(* CODESYS project ecomatDisplaytestIn2001.project
   Author: ifm electronic
   Version: 4.0.0.0
   Description: Project template for 4.3" ifm ecomat display  device with keypad.
   Title: ifm ecomatDisplay 4.3" 64bit with Keypad
   CompiledLibraryCompatibilityVersion: CODESYS V3.5 SP16 Patch 5
   Company: ifm electronic

Project tree, tasks and I/O mapping:
  Device : ecomatDisplay43inch_64bit, ifm electronic, version 3.5.19.72
    application Application
      libraries: ifm_ecomatDisplay43inch_Cnt, 1.1.0.0 (ifm electronic); ifmCANopenManager, * (ifm electronic); ifmRawCAN, * (ifm electronic); ifmBehavior, * (ifm electronic); ifmBehavior_ecomatDisplay, * (ifm electronic); ifmDevice_ecomatDisplay43inch, * (ifm electronic); ifmEcoSysLx_SysItf_Common, * (ifm electronic); ifmEcoSysLx_SysItf_Display, * (ifm electronic); ifmEcoSysLx_SysItf_IO, * (ifm electronic); ifmEcoSysLx_SysItf_Keypad, * (ifm electronic); ifmEcoSysLx_SysItf_Net, * (ifm electronic); ifmEcoSysLx_SysItf_Print, * (ifm electronic); ifmEcoSysLx_SysItf_RTC, * (ifm electronic); ifmEcoSysLx_SysItf_Service, * (ifm electronic); ifmEcoSysLx_SysItf_Storage, * (ifm electronic); ifmEcoSysLx_SysItf_SysInfo, * (ifm electronic); ifmEcoSysLx_SysItf_Touchscreen, * (ifm electronic); ifmFileUtil_ecomatDisplay, * (ifm electronic); ifmLLCAN, * (ifm electronic); ifmTypes, * (ifm electronic); ifmTypes_ecomatDisplay, * (ifm electronic); SM3_Basic, * (CODESYS); VisuSymbols, 4.5.0.0 (System); SysTimeCore, * (System); SysTimeRtc, * (System); SML_Basic, * (CODESYS); SM3_Ramps, * (3S - Smart Software Solutions GmbH); SysTypes Interfaces, * (System); Standard, 3.3.0.10 (System); Util, 3.5.19.0 (System); Standard64, 3.5.20.0 (System); BASIC, 3.31 (OSCAT); String Functions, 3.5.18.0 (3S - Smart Software Solutions GmbH)
      task VISU_TASK (cyclic, interval t#20ms, priority 15) calls VisuElems.Visu_Prg
      task Task (cyclic, interval 20 ms, priority 1) calls PLC_PRG
      task frame_control_1K500 (cyclic, interval t#20ms, priority 5) calls Main_FRAME_CONTROL
      GlobalVariables/
        global variables GVL_Buttons
        global variables GVL_PRG
        global variables GVL_KeyList
        global variables GVL_Sites
        Structs/
        global variables GVL_CAN
        global variables GVL_KeysConfig
        global variables Color
        data type ByteArray_t
      TextLists/
        text list TL_eKeyMapCodes
      image pool ifmImagePool
      FBs/
        location/
          function block locatoinSimulation [FBD]
        Paramater/
          function block TO_ArrayOfUsint [FBD]
          function block FB_ByteToBoolArray [FBD]
          function block FB_UpdatingDistanceParameter [FBD]
          function block parameterUpdate [FBD]
          function block PrepareParameterForCAN [FBD]
        Roboter_States/
          function block FB_CAN_TX_GetStates_Cyclic [FBD]
          function block FB_SoC_FromVoltage [ST]
        function block FB_DefineMotorControllerState [FBD]
        Controll/
          function block HMIControl [FBD]
          function block RoboterControl [FBD]
          function block AutomaticModeControl [FBD]
          function block SprayerControl [FBD]
        function block changeLanguage [FBD]
      image pool ImagePool
      Visu/
        visualisation Main_Site
        visualisation NewSiteFrame
        visualisation Srart_Site
        visualisation Roboter_Parameter
        visualisation Auto_Mode_Site
        visualisation Visu_Default
        visualisation keys_frame
        visualisation empty
      Programms/
        program PLC_PRG [FBD]: ACT_Errors_Handling, ACT_Setting, ACT_PressedKeysConfig, ACT_Button_Control
        program Main_FRAME_CONTROL [FBD]: ACT_FrameControl, ACT_RefreshhMI
      functions/
        function block FB_smoothCLK [FBD]
        function intToSelectOnBool [FBD]
        function block FB_CLK [FBD]
        function block Advanced_CTUD [FBD]
        function block fb_delay [FBD]
        function Stuffing_To_ArrayOfUsint [FBD]
        function F_AnyToByte [ST]
      can/
        function block FB_CAN_RX [FBD]
    Communication : Communication, ifm electronic, version 3.5.19.72
      Ethernet : Ethernet, ifm electronic, version 3.5.19.72
      CAN : CAN, ifm electronic, version 3.5.19.72
        CANbus : CANbus, ifm electronic, version 2.0.0.0
            settings: Baudrate = 500
  5ce3da45-db07-42e7-a21c-a00fff4ed8f6|E:\BSR\Me\May Be Useful\ifm-engg_Logo\IFMLO_PANT_2c.png
  5ce3da45-db07-42e7-a21c-a00fff4ed8f6|E:\BSR\OnSVN\CODESYS_V3x\PDM360-3\DesignDocs\Pictures\PDM Visu Templates 20181217\Bg_5Inch_dark.png
  5ce3da45-db07-42e7-a21c-a00fff4ed8f6|E:\BSR\OnSVN\CODESYS_V3x\PDM360-3\DesignDocs\Pictures\PDM Visu Templates 20181217\Bg_5Inch_lightPDM_Theming.png
  5ce3da45-db07-42e7-a21c-a00fff4ed8f6|E:\BSR\OnSVN\CODESYS_V3x\PDM360-3\DesignDocs\Pictures\PDM Visu Templates 20181217\Button_5Inch_dark.png
  5ce3da45-db07-42e7-a21c-a00fff4ed8f6|E:\BSR\OnSVN\CODESYS_V3x\PDM360-3\DesignDocs\Pictures\PDM Visu Templates 20181217\Button_5Inch_lightPDM_Theming.png
  5ce3da45-db07-42e7-a21c-a00fff4ed8f6|E:\BSR\OnSVN\CODESYS_V3x\PDM360-3\DesignDocs\Pictures\PDM Visu Templates 20181217\Button_And_Bg_5Inch_dark.png
  5ce3da45-db07-42e7-a21c-a00fff4ed8f6|E:\BSR\OnSVN\CODESYS_V3x\PDM360-3\DesignDocs\Pictures\PDM Visu Templates 20181217\Button_And_Bg_5Inch_lightPDM_Theming.png
  5ce3da45-db07-42e7-a21c-a00fff4ed8f6|C:\Users\indongpa\Downloads\Visu_KeyTemplates_ecomatDisplay43Inch_V2\LightBg_LightKey.png
  5ce3da45-db07-42e7-a21c-a00fff4ed8f6|C:\Users\indongpa\Downloads\Visu_KeyTemplates_ecomatDisplay43Inch_V2\WhiteBg_LightKey.png
  5ce3da45-db07-42e7-a21c-a00fff4ed8f6|C:\Users\indongpa\Downloads\Visu_Global_BG_ecomatDisplay43Inch_V1\Visu_Global_BG_NoKeys_ecomatDisplay43Inch.png
  5ce3da45-db07-42e7-a21c-a00fff4ed8f6|C:\Users\indongpa\OneDrive - ifm electronic gmbh\Downlaods\Visu_Global_BG_ecomatDisplay43Inch_V1\Visu_Global_BG_NoKeys_ecomatDisplay43Inch 90Deg.png
  5ce3da45-db07-42e7-a21c-a00fff4ed8f6|C:\Users\indongpa\Downloads\MicrosoftTeams-image (5).png
  5ce3da45-db07-42e7-a21c-a00fff4ed8f6|C:\Users\indongpa\Downloads\Visu_KeyTemplates_ecomatDisplay43Inch_V2\WhiteBg_DarkKey.png
  5ce3da45-db07-42e7-a21c-a00fff4ed8f6|C:\Users\indongpa\Downloads\Visu_Global_BG_ecomatDisplay43Inch_V1\Visu_Global_BG_WithKeys_ecomatDisplay43Inch.png
  5ce3da45-db07-42e7-a21c-a00fff4ed8f6|C:\Users\indongpa\Downloads\Visu_KeyTemplates_ecomatDisplay43Inch_V2\DarkBg_LightKey.png
  5ce3da45-db07-42e7-a21c-a00fff4ed8f6|C:\Users\indongpa\Downloads\Visu_KeyTemplates_ecomatDisplay43Inch_V2\Bg_Dark.png
  5ce3da45-db07-42e7-a21c-a00fff4ed8f6|C:\Users\indongpa\Downloads\Visu_KeyTemplates_ecomatDisplay43Inch_V2\Bg_Light.png
  Project Information/
    function GetCompany [ST]
    function GetTitle [ST]
    function GetVersion [ST]
    function GetTextProperty [ST]
    function GetTextProperty2 [ST]
    function GetNumberProperty [ST]
    function GetBooleanProperty [ST]
    function GetVersionProperty [ST]
  5ce3da45-db07-42e7-a21c-a00fff4ed8f6|C:\Users\indongpa\OneDrive - ifm electronic gmbh\Downlaods\Visu_Global_BG_ecomatDisplay43Inch_V1\Visu_Global_BG_WithKeys_ecomatDisplay43Inch 90Deg.png
  text list GlobalTextList
  5ce3da45-db07-42e7-a21c-a00fff4ed8f6|E:\BSR\Me\May Be Useful\ifm-engg_Logo\IFMLO_PANT_2c.png
  5ce3da45-db07-42e7-a21c-a00fff4ed8f6|C:\Users\indongpa\Downloads\Visu_KeyTemplates_ecomatDisplay43Inch_V2\DarkBg_LightKey.png
  5ce3da45-db07-42e7-a21c-a00fff4ed8f6|C:\Users\indongpa\Downloads\Visu_KeyTemplates_ecomatDisplay43Inch_V2\WhiteBg_DarkKey.png
  5ce3da45-db07-42e7-a21c-a00fff4ed8f6|C:\Users\indongpa\Downloads\Visu_KeyTemplates_ecomatDisplay43Inch_V2\LightBg_LightKey.png
  5ce3da45-db07-42e7-a21c-a00fff4ed8f6|C:\Users\indongpa\Downloads\Visu_KeyTemplates_ecomatDisplay43Inch_V2\WhiteBg_LightKey.png
  5ce3da45-db07-42e7-a21c-a00fff4ed8f6|C:\Users\indongpa\Downloads\Visu_Global_BG_ecomatDisplay43Inch_V1\Visu_Global_BG_WithKeys_ecomatDisplay43Inch.png
  5ce3da45-db07-42e7-a21c-a00fff4ed8f6|C:\Users\indongpa\OneDrive - ifm electronic gmbh\Downlaods\Visu_Global_BG_ecomatDisplay43Inch_V1\Visu_Global_BG_WithKeys_ecomatDisplay43Inch 90Deg.png
  5ce3da45-db07-42e7-a21c-a00fff4ed8f6|C:\Users\indongpa\Downloads\Visu_Global_BG_ecomatDisplay43Inch_V1\Visu_Global_BG_NoKeys_ecomatDisplay43Inch.png
  5ce3da45-db07-42e7-a21c-a00fff4ed8f6|C:\Users\indongpa\OneDrive - ifm electronic gmbh\Downlaods\Visu_Global_BG_ecomatDisplay43Inch_V1\Visu_Global_BG_NoKeys_ecomatDisplay43Inch 90Deg.png
  5ce3da45-db07-42e7-a21c-a00fff4ed8f6|C:\Users\indongpa\Downloads\Visu_KeyTemplates_ecomatDisplay43Inch_V2\Bg_Dark.png
  5ce3da45-db07-42e7-a21c-a00fff4ed8f6|C:\Users\indongpa\Downloads\Visu_KeyTemplates_ecomatDisplay43Inch_V2\Bg_Light.png
  5ce3da45-db07-42e7-a21c-a00fff4ed8f6|C:\Users\Administrator\Downloads\ant.png
  5ce3da45-db07-42e7-a21c-a00fff4ed8f6|C:\Users\Administrator\Downloads\Screenshot 2024-06-27 111636.png
  5ce3da45-db07-42e7-a21c-a00fff4ed8f6|C:\Users\Administrator\Downloads\Screenshot 2024-06-27 113436.png
  5ce3da45-db07-42e7-a21c-a00fff4ed8f6|C:\Users\moham\Downloads\splash_ant.bmp
  5ce3da45-db07-42e7-a21c-a00fff4ed8f6|C:\Users\Administrator\Downloads\ant_s.png
  5ce3da45-db07-42e7-a21c-a00fff4ed8f6|C:\Users\Administrator\Downloads\WhatsApp Image 2024-09-06 at 21.10.24.jpeg
  5ce3da45-db07-42e7-a21c-a00fff4ed8f6|C:\Users\Administrator\Downloads\battery fast Leer.png
  5ce3da45-db07-42e7-a21c-a00fff4ed8f6|C:\Users\Administrator\Downloads\images.jpg
  5ce3da45-db07-42e7-a21c-a00fff4ed8f6|C:\Users\Administrator\Downloads\304be42a-81d5-456b-8698-6dc5f69a8eec.jpg
  5ce3da45-db07-42e7-a21c-a00fff4ed8f6|C:\Users\Administrator\Downloads\269b2263-283b-4274-9266-790e9879ed38.jpg
  text list SwitchKeys
  5ce3da45-db07-42e7-a21c-a00fff4ed8f6|C:\Users\Administrator\Downloads\icons8-einstellung-50.png
  5ce3da45-db07-42e7-a21c-a00fff4ed8f6|C:\Users\Administrator\Downloads\battery_0.png
  5ce3da45-db07-42e7-a21c-a00fff4ed8f6|C:\Users\Administrator\Downloads\battery_10.png
  5ce3da45-db07-42e7-a21c-a00fff4ed8f6|C:\Users\Administrator\Downloads\battery_20.png
  5ce3da45-db07-42e7-a21c-a00fff4ed8f6|C:\Users\Administrator\Downloads\battery_30.png
  5ce3da45-db07-42e7-a21c-a00fff4ed8f6|C:\Users\Administrator\Downloads\battery_50.png
  5ce3da45-db07-42e7-a21c-a00fff4ed8f6|C:\Users\Administrator\Downloads\battery_70.png
  5ce3da45-db07-42e7-a21c-a00fff4ed8f6|C:\Users\Administrator\Downloads\battery_80.png
  5ce3da45-db07-42e7-a21c-a00fff4ed8f6|C:\Users\Administrator\Downloads\battery_90.png
  5ce3da45-db07-42e7-a21c-a00fff4ed8f6|C:\Users\Administrator\Downloads\battery_voll.png
  5ce3da45-db07-42e7-a21c-a00fff4ed8f6|C:\Users\moham\Downloads\ant(2).bmp
*)

// Device/Application/GlobalVariables/ByteArray_t
TYPE ByteArray_t : ARRAY[0..7] OF BYTE; END_TYPE

// Device/Application/GlobalVariables/GVL_Buttons
{attribute 'qualified_only'}
VAR_GLOBAL
	startAutoModeIsClicked: BOOL;
	stopAutoModeIsClicked: BOOL;
	//switschingToStartSite: BOOL;
	PauseAutoModeIsClicked: BOOL;
	backToStartScreenIsClicked: BOOL;
	settingClicked: BOOL;
	ResumeAutoModeIsClicked: BOOL;
	PauseOrResumeIsClicked: BOOL;
	
	
	// settings
		//time
		
// parameter
	//start time
	//sprayer
	sprayerUp : BOOL;
	sprayerDown : BOOL;
	sprayerLeft : BOOL;
	sprayerRight : BOOL;
	pump : BOOL;
	//Language
	englisch: BOOL;
	deutsch: BOOL;
	//changeHourClicked: BOOL;
	//changeMinuteClicked: BOOL;
END_VAR

// Device/Application/GlobalVariables/GVL_PRG
{attribute 'qualified_only'}
VAR_GLOBAL

	// HMI Mode
	deactivatePLCSimModeMan: BOOL;
	// visu frames control
	currentVisuFrame: INT := 0;
	refreshHMI : BOOL := FALSE; // use rising/falling trigger
	
	//parameter
	selectedParameterIndex: Int:= 0;
	bRowsDirection: BOOL;
	rCountRows: REAL;
	roboterWidth: REAL:= 0.5;
	dinstanceBetweenRowsMin: REAL := roboterWidth + 0.2; // m : min. distance between 2 Rows in meter. Ther is no max Value but the max Value is in CAN Frame for all distances d1,d2 and d3 = 12.8 m  
	turningDistancerMin: REAL:= 1.5; // min distance to be able to make a turn
	
	// Automode Control
	SR_autoMode: SR;
	RS_AM_Paused: RS;
	AM_Paused: BOOL;
	autoModestarted: BOOL;
	screenSwitching: BOOL;	// while switching the frame: true to disable all buttons
	enableAM : BOOL := TRUE;
	//State
	batteryState: USINT;
	enableStatesRequest : BOOL := TRUE;
	
	
	activate_FrameControl : BOOL := TRUE;
	
	//Sprayer
	
	enableSprayer : BOOL := TRUE;
	
	// CAN
	
	enableCanChannel_0: BOOL;
	canInfo: ifmTypes.DIAG_INFO;
	restartCan: BOOL;
	sprayerCanInfo: ifmTypes.DIAG_INFO;
	sprayerCanError: BOOL;
	canChannelError: BOOL;
	AM_CanFramError: BOOL;
	canError: BOOL;
	stetesCanError: BOOL;
	deactivateErrorHandling: BOOL;
	SR_startIsKlicked: SR;
	startMin: INT;
	startHour: INT;
	waitingStartTime: BOOL;
	simModeActive: BOOL;
	stopAM_Frame_received: BOOL;
	showkeys: BOOL;
	frameid: USINT;
	frameRefreshRequestCanError: BOOL;
	canFatalError: BOOL;
	fatalErrot: BOOL;
	to_am_frame: BOOL;
	stTime: ifmDevice.stDATE_TIME;
	acceleration: UINT;
	accelerationX10: UDINT;
	deceleration: UINT;
	decelerationX10: UDINT;
	settingCanError: BOOL;
	accelerationScreen: UINT;
	decelerationScreen: UINT;
END_VAR
VAR_GLOBAL RETAIN
	// setting
	language : STRING := 'EN';
	maxVoltage : REAL := 58.4;
	sprayerHight : REAL;
	MotorSpeed : USINT;
END_VAR
VAR_GLOBAL CONSTANT
		allwaysTrue : BOOL := TRUE;
END_VAR

// Device/Application/GlobalVariables/GVL_KeyList
{attribute 'qualified_only'}

(* 

!!! This GVL list is from project template !!!

The following variables are controlled by key events mapped at Default Hotkey mapping list in Visualization Manager.

For example, F1 function key of standard keyboard (MFII) is pressed, xF1 bit in this list will become TRUE; when the same 
key is released then xF1 become FALSE.

*)

VAR_GLOBAL

(* Display system key press / release event status. TRUE = Key Pressed, FALSE = Key Released  *)
	xF1 		: BOOL;		(* Event status of F1 function key *)
	xF2 		: BOOL;		(* Event status of F2 function key *)
	xF3 		: BOOL;		(* Event status of F3 function key *)
	xF4 		: BOOL;		(* Event status of F4 function key *)
	xF5 		: BOOL;		(* Event status of F5 function key *)
	xF6 		: BOOL;		(* Event status of F6 function key *)
	xF7 		: BOOL;		(* Event status of F7 function key *)
	xF8 		: BOOL;		(* Event status of F8 function key *)
	xF9 		: BOOL;		(* Event status of F9 function key *)
	xF10 		: BOOL;		(* Event status of F10 function key *)
	xUp 		: BOOL;		(* Event status of Up arrow key *)
	xDown		: BOOL;		(* Event status of Down arrow key *)
	xLeft 		: BOOL;		(* Event status of Left arrow key *)
	xRight 		: BOOL;		(* Event status of Right arrow key *)
	xKey_Return : BOOL;		(* Event status of Return (or Enter) key *)
END_VAR

// Device/Application/GlobalVariables/GVL_Sites
{attribute 'qualified_only'}
VAR_GLOBAL
	Parameter:STRING:= 'Roboter_Parameter';
	location: STRING:= 'LocationSeite_Inkrement';
END_VAR

// Device/Application/GlobalVariables/GVL_CAN
{attribute 'qualified_only'}
VAR_GLOBAL
	
	canChannnel: ifmDevice.CAN_CHANNEL := ifmDevice.CAN_CHANNEL.CHAN_0;
	// States ID 16x601
	getStatusState: ARRAY [0..7] OF USINT := [16#40,16#11,16#21,0,0,0,0,0];
	getFaultsState: ARRAY [0..7] OF USINT := [16#40,16#12,16#21,0,0,0,0,0];
	getBatteryState: ARRAY [0..7] OF USINT := [16#42,16#0D,16#21,2,0,0,0,0];
	getRuntimeStatus1: ARRAY [0..7] OF USINT := [16#40,16#22,16#21,1,0,0,0,0]; //1. Motor Andrew needs to change 1 and 2
	getRuntimeStatus2: ARRAY [0..7] OF USINT := [16#40,16#22,16#21,2,0,0,0,0]; //2. Motor
	
	// auto Mode
	automodeCanId: UDINT := 16#50;
	
	stop: ARRAY [0..7] OF USINT:=[255,0,0,0,0,0,0,0];
	pause: ARRAY [0..7] OF USINT:=[200,1,0,0,0,0,0,0];
	resume: ARRAY [0..7] OF USINT:=[200,2,0,0,0,0,0,0];
	
	// acceleration Profile
	//getAcceleration_1: ARRAY [0..7] OF USINT:=[16#40,16#83,16#60,1,0,0,0,0];
	//setAcceleration_1: ARRAY [0..7]OF USINT:=[16#40,16#83,16#60,1,0,0,0,0];
	//getDeceleration_1: ARRAY [0..7] OF USINT:=[16#40,16#84,16#60,1,0,0,0,0];
	//setDeceleration_1: ARRAY [0..7] OF USINT:=[16#40,16#07,16#20,1,0,0,0,0];
	
	//getAcceleration_2: ARRAY [0..7] OF USINT:=[16#40,16#83,16#60,1,0,0,0,0];
	//setAcceleration_2: ARRAY [0..7] OF USINT:=[16#40,16#08,16#20,1,0,0,0,0];
	//getDeceleration_2: ARRAY [0..7] OF USINT:=[16#40,16#84,16#60,1,0,0,0,0];
	//setDeceleration_2: ARRAY [0..7] OF USINT:=[16#40,16#07,16#20,1,0,0,0,0];
	//setAcceleration_1: ARRAY [0..7] OF USINT:=[16#40,16#08,16#20,1,0,0,0,0];
	
	// acceleration Value
	setAcceleration_1: ARRAY [0..7]OF USINT:=[16#23,16#06,16#20,1,0,0,0,0];
	setAcceleration_2: ARRAY [0..7]OF USINT:=[16#23,16#06,16#20,2,0,0,0,0];
	setDeceleration_1: ARRAY [0..7]OF USINT:=[16#23,16#07,16#20,1,0,0,0,0];
	setDeceleration_2: ARRAY [0..7]OF USINT:=[16#23,16#07,16#20,2,0,0,0,0];
	
	// max. rpm
	setRPM_max_1 :ARRAY [0..7]OF USINT:=[16#23,16#07,16#20,1,0,0,0,0];
	// get motors data
	reedRPM: ARRAY [0..7] OF USINT:=[16#40,16#03,16#21,1,0,0,0,0];// Min: -65535  Max: 65535
	Read_Battery_Amps : ARRAY [0..7] OF USINT:=[16#42,16#0C,16#21,1,0,0,0,0]; // Measures and reports the Amps flowing from the battery in Amps * 10
	Read_Battery_State_Of_Charge : ARRAY [0..7] OF USINT:=[16#42,16#3A,16#21,0,0,0,0,0]; // Battery state of charge in %
	//Sprayer
	
	motorcontrollerId: UDINT := 16#601;
	
	//control some of bits
	switchOffPump: ARRAY [0..7] OF USINT:=[16#2F,16#0A,16#20,0,6,0,0,0];
	switchOnPump: ARRAY [0..7] OF USINT:=[16#2F,16#09,16#20,0,6,0,0,0];
	switchOffSprayerLeft: ARRAY [0..7] OF USINT:=[16#2F,16#0A,16#20,0,7,0,0,0];
	switchOnSprayerLeft: ARRAY [0..7] OF USINT:=[16#2F,16#09,16#20,0,7,0,0,0];
	switchOffSprayerRight: ARRAY [0..7] OF USINT:=[16#2F,16#0A,16#20,0,8,0,0,0];
	switchOnSprayerRight: ARRAY [0..7] OF USINT:=[16#2F,16#09,16#20,0,8,0,0,0];
	sprayeStartUpFrame: ARRAY [0..7] OF USINT:=[47,9,32,0,2,0,0,0];// Andrew: 4->1 & -4->2 when paused & stop
	sprayerStopUpFrame: ARRAY [0..7] OF USINT:=[47,10,32,0,2,0,0,0];// When resume 4->1 & 2
	sprayerStartDownFrame: ARRAY [0..7] OF USINT:=[47,9,32,0,4,0,0,0];
	sprayerStopDownFrame: ARRAY [0..7] OF USINT:=[47,10,32,0,4,0,0,0];
	
	HMI_CAN_ID: UDINT := 16#19;
	ACK_Stop : ARRAY [0..7] OF USINT:=[3,0,0,0,0,0,0,0];
	stopFrameJetson : ARRAY [0..7] OF USINT :=[2,0,0,0,0,0,0,0];
	test: ARRAY [0..7] OF USINT := [8(1)];
END_VAR

// Device/Application/GlobalVariables/GVL_KeysConfig
{attribute 'qualified_only'}
VAR_GLOBAL
	countOfPressedKeys : USINT;
	oneKeyPressedForLongTime: BOOL;
	oneKeyOrMorePressed: BOOL;
	oneKeyPressed: BOOL;
	oneKeyPressedForLongTime_RT: BOOL;
END_VAR

// Device/Application/GlobalVariables/Color

{attribute 'qualified_only'}
VAR_GLOBAL
	
	NOT_DEFINED : DINT :=-1;
	Aqua : DINT :=16#FFFF;
	Black : DINT :=16#0;
	Blue : DINT :=16#FF;
	Brown : DINT :=16#A52A2A;
	Cyan : DINT :=16#FFFF;
	DarkBlue : DINT :=16#8B;
	DarkCyan : DINT :=16#8B8B;
	DarkGray : DINT :=16#A9A9A9;
	DarkGreen :DINT :=16#6400;
	DarkMagenta : DINT :=16#8B008B; 
	DarkRed : DINT :=16#8B0000;
	DimGray :DINT :=16#696969;
	Gray : DINT :=16#808080;
	Green : DINT :=16#8000;
	LightBlue : DINT :=16#ADD8E6;
	LightCyan : DINT :=16#E0FFFF;
	LightGray : DINT :=16#D3D3D3;
	LightGreen : DINT :=16#90EE90;
	LightYellow : DINT :=16#FFFFE0;
	Lime : DINT :=16#FF00;
	Magenta : DINT :=16#FF00FF;
	Maroon : DINT :=16#800000;
	Navy : DINT :=16#80;
	Olive : DINT :=16#808000;
	Purple : DINT :=16#800080;
	Red : DINT  :=16#FF0000;
	Silver : DINT :=16#C0C0C0;
	Teal : DINT :=16#8080;
	White : DINT :=16#FFFFFF;
	Yellow : DINT := 16#FFFF00;
	
	// Transperancy
	TRANSP_NO : BYTE := 16#FF;
	TRANSP_LOW : BYTE := 16#C0;
	TRANSP_MEDIUM : BYTE := 16#80;
	TRANSP_HIGH : BYTE := 16#40;
	TRANSP_FULL  : BYTE := 16#0;

	batteryColor : DINT := 16#8000;
	keysColor: UDINT := 16#FF6E00;

END_VAR

// Device/Application/Programms/PLC_PRG

(* !!! This POU is from project template !!! *)

PROGRAM PLC_PRG
VAR
	testframe: ARRAY [0..7] OF USINT := [16#40,16#11,16#21,0,0,0,0,0];
	canTestFrameTon : TON;
	RS_Test : RS;
	t_test : TIME := T#3000ms;
(* Below is the FB instance with initial values to set default key mapping. The default key map is as per the default values set for ifmDevice.stKEY_MAP_LIST. *)
	fbSetKeyMapping		: ifmDevice.SetKeyMapping;
	batteryStateInProcent: REAL;
	selectedParameterIndex: INT;
	FB_CAN_RX_0: FB_CAN_RX;
	FB_CAN_TX_GetStates_Cyclic_0: FB_CAN_TX_GetStates_Cyclic;
	FB_HMIControl_0: HMIControl;
	getUpdatedParameter: parameterUpdate;
	RoboterautoModeControl_0: RoboterControl;
	SprayerControl_0: SprayerControl;
	//locatoinSimulation_0: locatoinSimulation;
	CAN_Tx_0: ifmRCAN.CAN_Tx;

	keyDelay: TON := (PT := TIME#300MS);

	goToParameterFrame: BOOL;
	
	// ERRORS handling
	RS_DisableCan: Standard.RS;
	TON_CanDisabled: Standard.TON ;
	test: BOOL;
	ctu_restart_counter: Standard.CTU;
	SR_simModeActive: SR;
	usiNumberRetryCanRecover: USINT := 5;
	rs_canrec: rs;
	restartRecovery: BOOL;
	testAfterRecover: FB_clk;
	resetErrors: BOOL;
	Advanced_CTUD_changeSysTimeMin: Advanced_CTUD;
	Advanced_CTUD_changeSysTimeHour: Advanced_CTUD;
	test2: UINT;
	test3: ByteArray_t;
	acceleration: UDINT;
	ChangingAcceleration_0: Advanced_CTUD;
	CAN_Tx_setAcceleration_1: ifmRCAN.CAN_Tx;
	ChangingDeceleration_0: Advanced_CTUD;
	CAN_Tx_setDeceleration_1: ifmRCAN.CAN_Tx;
	CAN_Tx_setDeceleration_2: ifmRCAN.CAN_Tx;
	CAN_Tx_setAcceleration_2: ifmRCAN.CAN_Tx;
	TON_F1: TON;
	TON_F3: TON;
END_VAR
// setting
VAR
	currentSettingFrameId : SINT := 0;
	//currentMaxRows : USINT := 0;

	//countOfSeconderyMeneuRows2 : ARRAY [0 .. countOfSettingRows] OF SINT:= [0,0,1];
	//
	//EN: BOOL ;
	DE : BOOL ;
	RO : BOOL ;
	changeLanguage_EN: changeLanguage;
	changeLanguage_DE: changeLanguage;
	//mainMeneuActive : BOOL := TRUE;
	
	SR_DeactivateLeftMeneu: SR;
	deactivateMainMeneu: BOOL;
	deactivateSeconderyMeneu: BOOL;
	selectedRowNum_Right: SINT := 0;//-1;
	selectedRowNum_left: SINT  := 0;//-1;
	SR_Enable: SR;
	enable: BOOL := TRUE;
	SR_activate3rdColumn: SR;
	thirdColumnActive: BOOL;
	visuhelp : BOOL;
	TON_Delay: TON := (PT := TIME#105ms);
	selectedRowNum_Right2: SINT;
	RS_visuHelp2: RS;
	RS_visuHelp3: RS;
	RS_visuHelp4: RS;
	pumpOn: BOOL;
	RS_pump: RS;
	sprayerSelectionLimit: SINT;
	languageselectionLimit : SINT;
	TOGGLE_Pump: TOGGLE;
	hourSetting: UINT;
	settedHoursNow: UINT;
	setTime: BOOL;
	SetSysTime: ifmDevice.SetSysTime;
	newTime: ifmDevice.stDATE_TIME;
	CAN_Recover_0 : ifmRCAN.CAN_Recover;
END_VAR
VAR CONSTANT
	countOfSettingRows: SINT := 1;
	sprayerId : USINT := 1;
	languageID : USINT := 0;
	timeId: USINT := 2;
	countOfSeconderyMeneuRows : ARRAY [0 .. countOfSettingRows] OF SINT:= [1,4];
END_VAR

//button control
VAR
	startTime : TIME_OF_DAY;
	TON_StopresumeButtonVisible: ton;
	StopresumeButtonVisible: BOOL;
END_VAR
VAR // added by the converter: edge detectors and wires of the graphical bodies
    _rt1, _rt2, _rt3, _rt4, _rt5, _rt6, _rt7, _rt8, _rt9, _rt10, _rt11, _rt12, _rt13, _rt14, _rt15, _rt16, _rt17, _rt18, _rt19, _rt20, _rt21, _rt22, _rt23, _rt24, _rt25 : R_TRIG;
    _ft1, _ft2, _ft3, _ft4, _ft5, _ft6, _ft7, _ft8 : F_TRIG;
    _w1, _w2, _w3 : BOOL;
    _w4, _w5, _w6, _w7, _w8, _w9, _w10, _w11 : USINT;
END_VAR

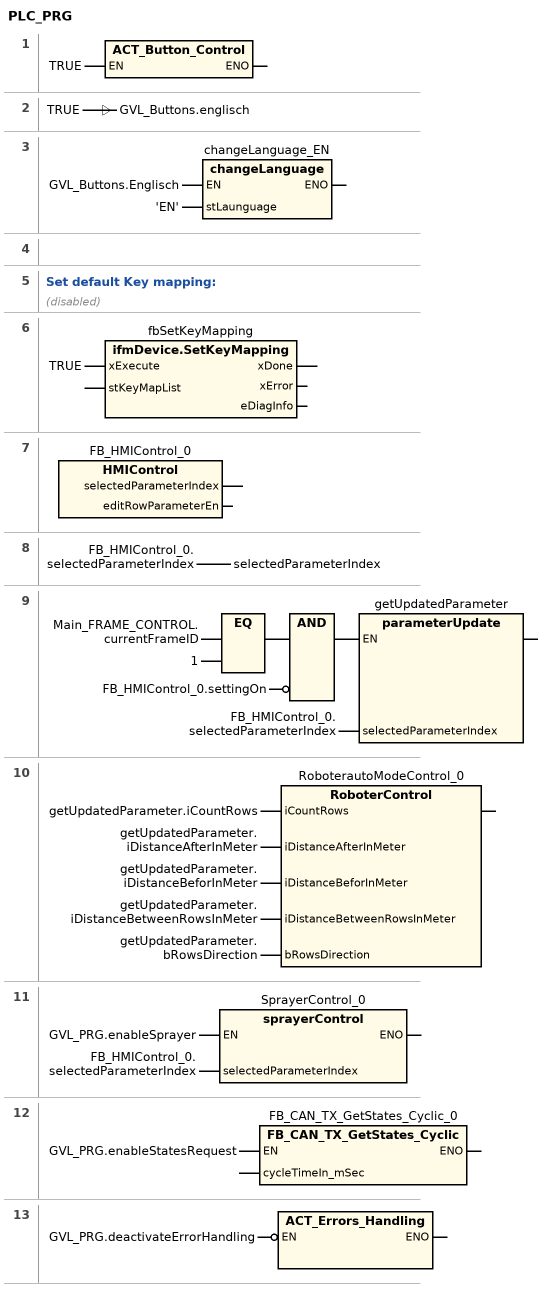
// NETWORK 1
ACT_Button_Control();

// NETWORK 2
_rt1(CLK := TRUE);
GVL_Buttons.englisch := _rt1.Q;

// NETWORK 3
IF GVL_Buttons.Englisch THEN
    changeLanguage_EN(stLaunguage := 'EN'); // changeLanguage
END_IF

// NETWORK 4

// NETWORK 5 (disabled)
// label: Set default Key mapping

// NETWORK 6
fbSetKeyMapping(xExecute := TRUE); // ifmDevice.SetKeyMapping

// NETWORK 7
FB_HMIControl_0(); // HMIControl

// NETWORK 8
selectedParameterIndex := FB_HMIControl_0.selectedParameterIndex;

// NETWORK 9
getUpdatedParameter(EN := Main_FRAME_CONTROL.currentFrameID = 1 AND NOT FB_HMIControl_0.settingOn, selectedParameterIndex := FB_HMIControl_0.selectedParameterIndex); // parameterUpdate

// NETWORK 10
RoboterautoModeControl_0(
    iCountRows := getUpdatedParameter.iCountRows,
    iDistanceAfterInMeter := getUpdatedParameter.iDistanceAfterInMeter,
    iDistanceBeforInMeter := getUpdatedParameter.iDistanceBeforInMeter,
    iDistanceBetweenRowsInMeter := getUpdatedParameter.iDistanceBetweenRowsInMeter,
    bRowsDirection := getUpdatedParameter.bRowsDirection); // RoboterControl

// NETWORK 11
IF GVL_PRG.enableSprayer THEN
    SprayerControl_0(selectedParameterIndex := FB_HMIControl_0.selectedParameterIndex); // sprayerControl
END_IF

// NETWORK 12
IF GVL_PRG.enableStatesRequest THEN
    FB_CAN_TX_GetStates_Cyclic_0(); // FB_CAN_TX_GetStates_Cyclic
END_IF

// NETWORK 13
IF NOT GVL_PRG.deactivateErrorHandling THEN ACT_Errors_Handling(); END_IF

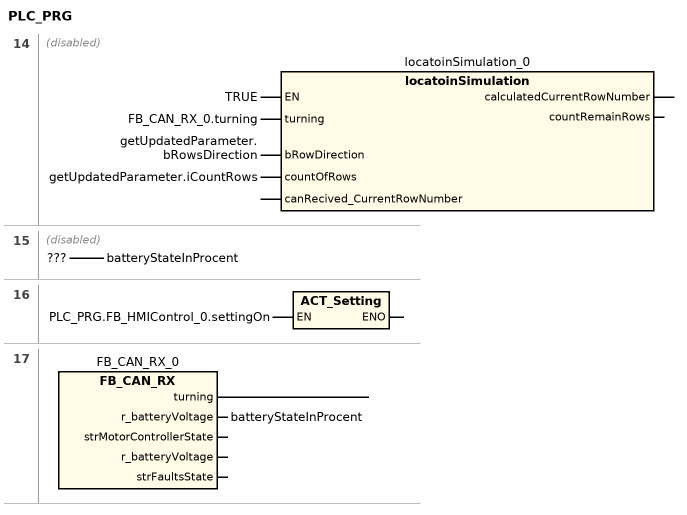
// NETWORK 14 (disabled)
// locatoinSimulation_0(
//     EN := TRUE,
//     turning := FB_CAN_RX_0.turning,
//     bRowDirection := getUpdatedParameter.bRowsDirection,
//     countOfRows := getUpdatedParameter.iCountRows); // locatoinSimulation

// NETWORK 15 (disabled)
// batteryStateInProcent := ???;

// NETWORK 16
IF PLC_PRG.FB_HMIControl_0.settingOn THEN ACT_Setting(); END_IF

// NETWORK 17
FB_CAN_RX_0(r_batteryVoltage => batteryStateInProcent); // FB_CAN_RX

ACTION ACT_Errors_Handling:
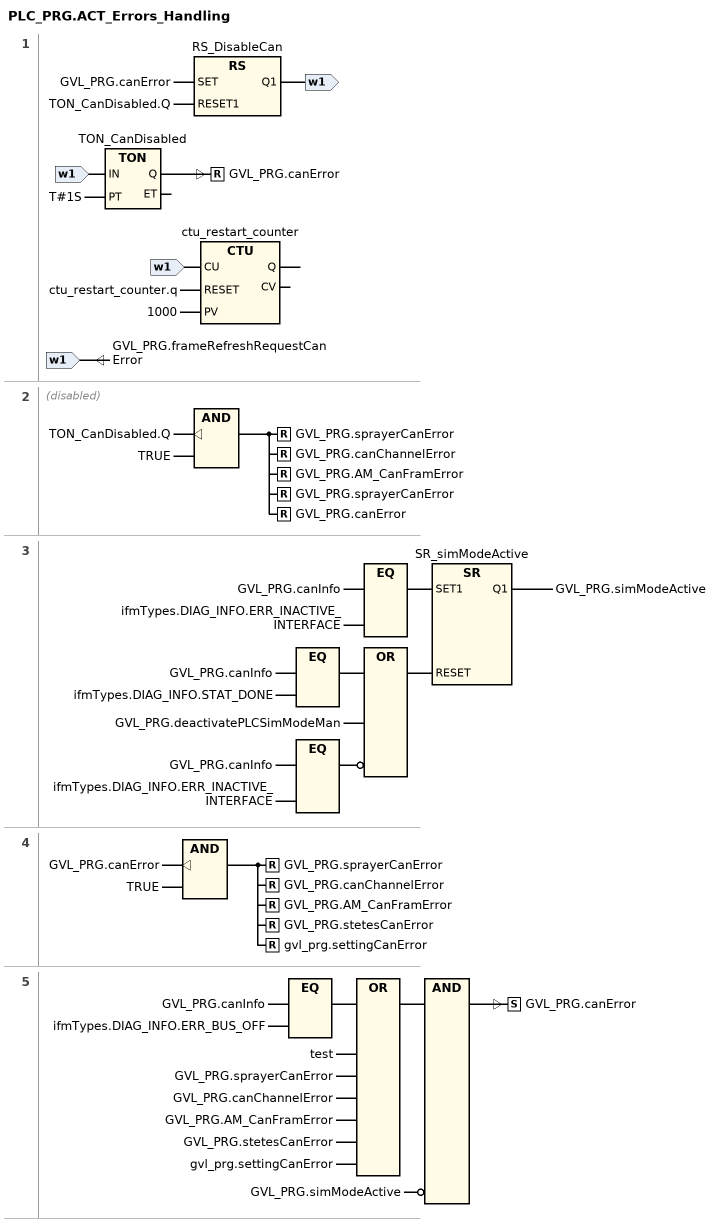
// NETWORK 1
RS_DisableCan(SET := GVL_PRG.canError, RESET1 := TON_CanDisabled.Q); // RS
TON_CanDisabled(IN := RS_DisableCan.Q1, PT := T#1S); // TON
_rt2(CLK := TON_CanDisabled.Q);
GVL_PRG.canError R= _rt2.Q;
ctu_restart_counter(CU := RS_DisableCan.Q1, RESET := ctu_restart_counter.q, PV := 1000); // CTU
_ft1(CLK := RS_DisableCan.Q1);
GVL_PRG.frameRefreshRequestCanError := _ft1.Q;

// NETWORK 2 (disabled)
// _ft2(CLK := TON_CanDisabled.Q);
// _w1 := _ft2.Q AND TRUE;
// GVL_PRG.sprayerCanError R= _w1;
// GVL_PRG.canChannelError R= _w1;
// GVL_PRG.AM_CanFramError R= _w1;
// GVL_PRG.sprayerCanError R= _w1;
// GVL_PRG.canError R= _w1;

// NETWORK 3
SR_simModeActive(SET1 := GVL_PRG.canInfo = ifmTypes.DIAG_INFO.ERR_INACTIVE_INTERFACE, RESET := GVL_PRG.canInfo = ifmTypes.DIAG_INFO.STAT_DONE OR GVL_PRG.deactivatePLCSimModeMan OR NOT (GVL_PRG.canInfo = ifmTypes.DIAG_INFO.ERR_INACTIVE_INTERFACE)); // SR
GVL_PRG.simModeActive := SR_simModeActive.Q1;

// NETWORK 4
_ft3(CLK := GVL_PRG.canError);
_w2 := _ft3.Q AND TRUE;
GVL_PRG.sprayerCanError R= _w2;
GVL_PRG.canChannelError R= _w2;
GVL_PRG.AM_CanFramError R= _w2;
GVL_PRG.stetesCanError R= _w2;
gvl_prg.settingCanError R= _w2;

// NETWORK 5
_rt3(CLK := (GVL_PRG.canInfo = ifmTypes.DIAG_INFO.ERR_BUS_OFF OR test OR GVL_PRG.sprayerCanError OR GVL_PRG.canChannelError OR GVL_PRG.AM_CanFramError OR GVL_PRG.stetesCanError OR gvl_prg.settingCanError) AND NOT GVL_PRG.simModeActive);
GVL_PRG.canError S= _rt3.Q;

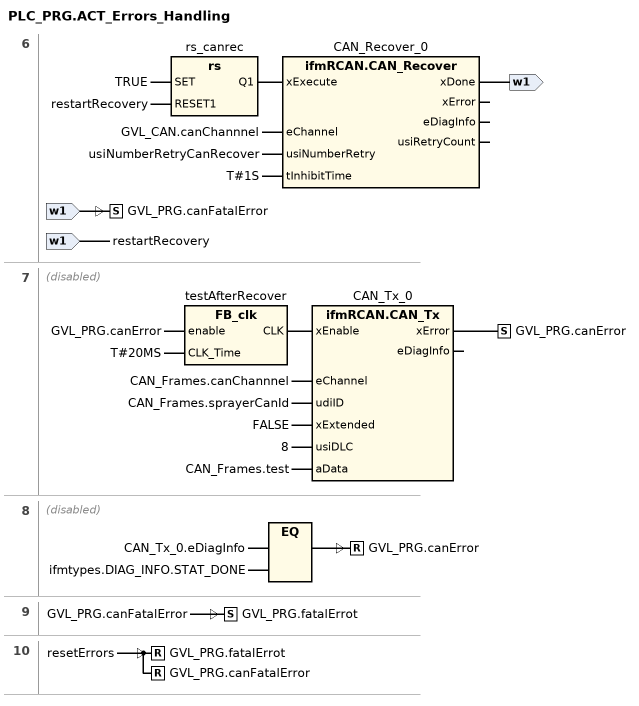
// NETWORK 6
rs_canrec(SET := TRUE, RESET1 := restartRecovery); // rs
CAN_Recover_0(
    xExecute := rs_canrec.Q1,
    eChannel := GVL_CAN.canChannnel,
    usiNumberRetry := usiNumberRetryCanRecover,
    tInhibitTime := T#1S); // ifmRCAN.CAN_Recover
_rt4(CLK := CAN_Recover_0.xDone);
GVL_PRG.canFatalError S= _rt4.Q;
restartRecovery := CAN_Recover_0.xDone;

// NETWORK 7 (disabled)
// testAfterRecover(enable := GVL_PRG.canError, CLK_Time := T#20MS); // FB_clk
// CAN_Tx_0(
//     xEnable := testAfterRecover.CLK,
//     eChannel := CAN_Frames.canChannnel,
//     udiID := CAN_Frames.sprayerCanId,
//     xExtended := FALSE,
//     usiDLC := 8,
//     aData := CAN_Frames.test); // ifmRCAN.CAN_Tx
// GVL_PRG.canError S= CAN_Tx_0.xError;

// NETWORK 8 (disabled)
// _rt5(CLK := CAN_Tx_0.eDiagInfo = ifmtypes.DIAG_INFO.STAT_DONE);
// GVL_PRG.canError R= _rt5.Q;

// NETWORK 9
_rt6(CLK := GVL_PRG.canFatalError);
GVL_PRG.fatalErrot S= _rt6.Q;

// NETWORK 10
_rt7(CLK := resetErrors);
GVL_PRG.fatalErrot R= _rt7.Q;
GVL_PRG.canFatalError R= _rt7.Q;
END_ACTION

ACTION ACT_Setting:
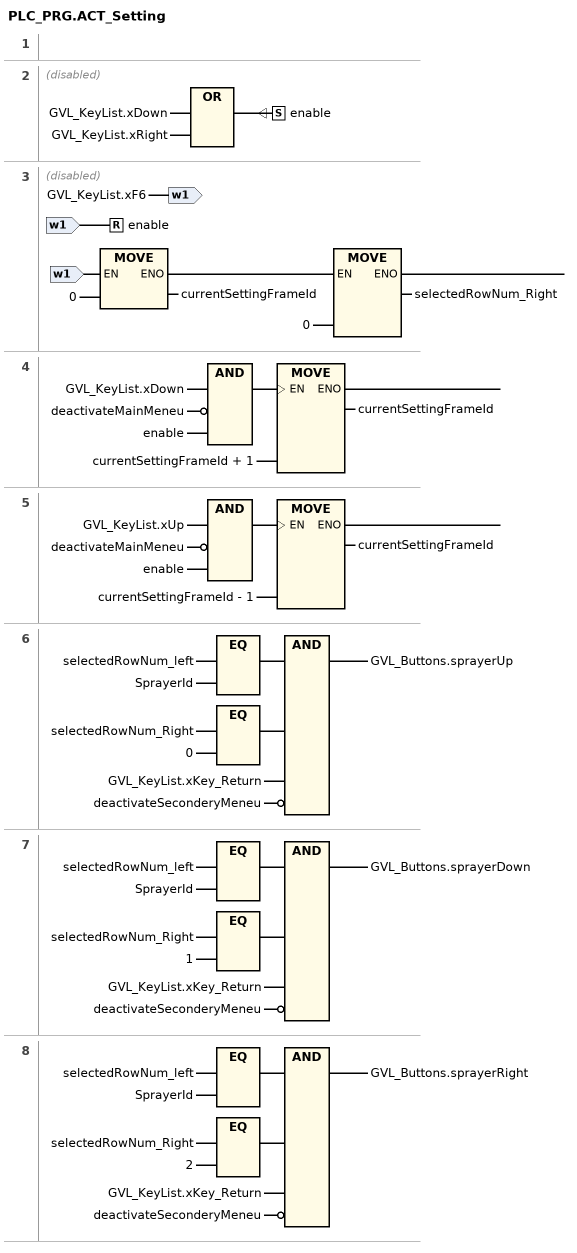
// NETWORK 1

// NETWORK 2 (disabled)
// _ft4(CLK := GVL_KeyList.xDown OR GVL_KeyList.xRight);
// enable S= _ft4.Q;

// NETWORK 3 (disabled)
// _rt8(CLK := GVL_KeyList.xF6);
// enable R= _rt8.Q;
// _w3 := _rt8.Q;
// IF _w3 THEN currentSettingFrameId := 0; END_IF
// IF _w3 THEN selectedRowNum_Right := 0; END_IF

// NETWORK 4
_rt9(CLK := GVL_KeyList.xDown AND NOT deactivateMainMeneu AND enable);
IF _rt9.Q THEN currentSettingFrameId := currentSettingFrameId + 1; END_IF

// NETWORK 5
_rt10(CLK := GVL_KeyList.xUp AND NOT deactivateMainMeneu AND enable);
IF _rt10.Q THEN currentSettingFrameId := currentSettingFrameId - 1; END_IF

// NETWORK 6
GVL_Buttons.sprayerUp := selectedRowNum_left = SprayerId AND selectedRowNum_Right = 0 AND GVL_KeyList.xKey_Return AND NOT deactivateSeconderyMeneu;

// NETWORK 7
GVL_Buttons.sprayerDown := selectedRowNum_left = SprayerId AND selectedRowNum_Right = 1 AND GVL_KeyList.xKey_Return AND NOT deactivateSeconderyMeneu;

// NETWORK 8
GVL_Buttons.sprayerRight := selectedRowNum_left = SprayerId AND selectedRowNum_Right = 2 AND GVL_KeyList.xKey_Return AND NOT deactivateSeconderyMeneu;

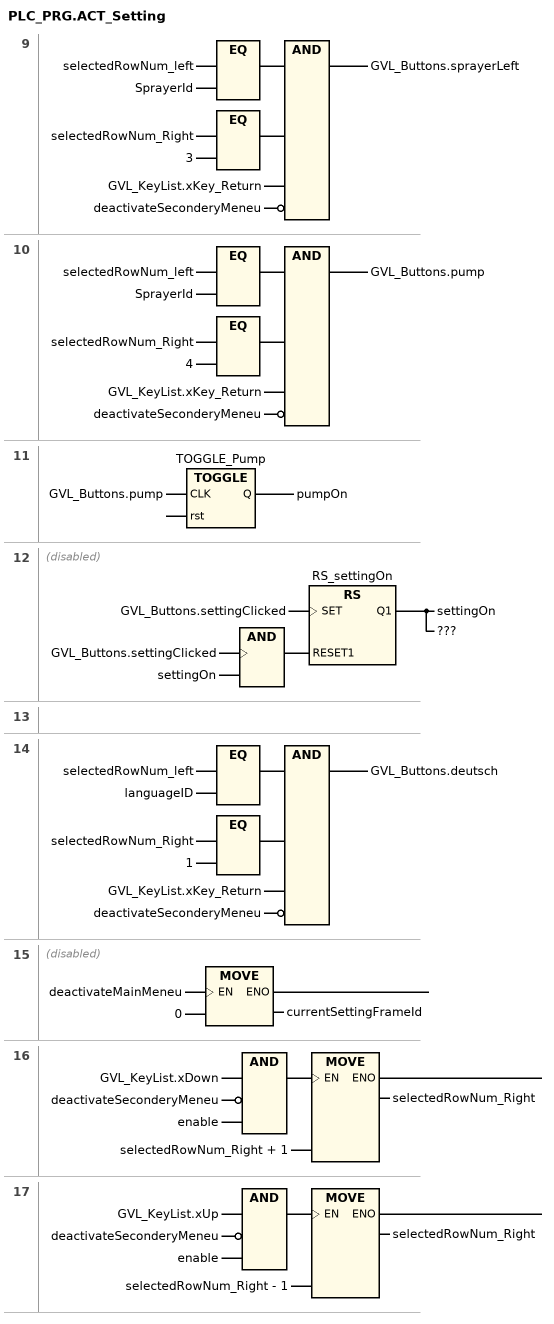
// NETWORK 9
GVL_Buttons.sprayerLeft := selectedRowNum_left = SprayerId AND selectedRowNum_Right = 3 AND GVL_KeyList.xKey_Return AND NOT deactivateSeconderyMeneu;

// NETWORK 10
GVL_Buttons.pump := selectedRowNum_left = SprayerId AND selectedRowNum_Right = 4 AND GVL_KeyList.xKey_Return AND NOT deactivateSeconderyMeneu;

// NETWORK 11
TOGGLE_Pump(CLK := GVL_Buttons.pump); // TOGGLE
pumpOn := TOGGLE_Pump.Q;

// NETWORK 12 (disabled)
// _rt11(CLK := GVL_Buttons.settingClicked);
// _rt12(CLK := GVL_Buttons.settingClicked);
// RS_settingOn(SET := _rt11.Q, RESET1 := _rt12.Q AND settingOn); // RS
// settingOn := RS_settingOn.Q1;
// ??? := RS_settingOn.Q1;

// NETWORK 13

// NETWORK 14
GVL_Buttons.deutsch := selectedRowNum_left = languageID AND selectedRowNum_Right = 1 AND GVL_KeyList.xKey_Return AND NOT deactivateSeconderyMeneu;

// NETWORK 15 (disabled)
// _rt13(CLK := deactivateMainMeneu);
// IF _rt13.Q THEN currentSettingFrameId := 0; END_IF

// NETWORK 16
_rt14(CLK := GVL_KeyList.xDown AND NOT deactivateSeconderyMeneu AND enable);
IF _rt14.Q THEN selectedRowNum_Right := selectedRowNum_Right + 1; END_IF

// NETWORK 17
_rt15(CLK := GVL_KeyList.xUp AND NOT deactivateSeconderyMeneu AND enable);
IF _rt15.Q THEN selectedRowNum_Right := selectedRowNum_Right - 1; END_IF

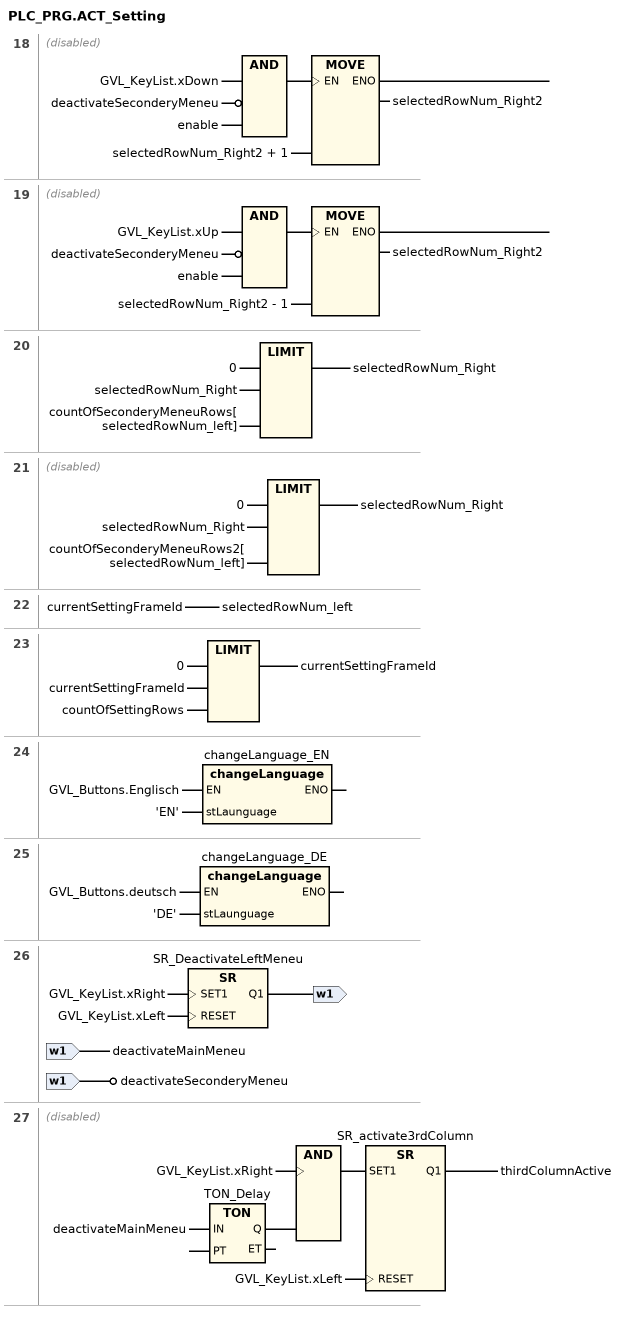
// NETWORK 18 (disabled)
// _rt16(CLK := GVL_KeyList.xDown AND NOT deactivateSeconderyMeneu AND enable);
// IF _rt16.Q THEN selectedRowNum_Right2 := selectedRowNum_Right2 + 1; END_IF

// NETWORK 19 (disabled)
// _rt17(CLK := GVL_KeyList.xUp AND NOT deactivateSeconderyMeneu AND enable);
// IF _rt17.Q THEN selectedRowNum_Right2 := selectedRowNum_Right2 - 1; END_IF

// NETWORK 20
selectedRowNum_Right := LIMIT(0, selectedRowNum_Right, countOfSeconderyMeneuRows[selectedRowNum_left]);

// NETWORK 21 (disabled)
// selectedRowNum_Right := LIMIT(0, selectedRowNum_Right, countOfSeconderyMeneuRows2[selectedRowNum_left]);

// NETWORK 22
selectedRowNum_left := currentSettingFrameId;

// NETWORK 23
currentSettingFrameId := LIMIT(0, currentSettingFrameId, countOfSettingRows);

// NETWORK 24
IF GVL_Buttons.Englisch THEN
    changeLanguage_EN(stLaunguage := 'EN'); // changeLanguage
END_IF

// NETWORK 25
IF GVL_Buttons.deutsch THEN
    changeLanguage_DE(stLaunguage := 'DE'); // changeLanguage
END_IF

// NETWORK 26
_rt18(CLK := GVL_KeyList.xRight);
_rt19(CLK := GVL_KeyList.xLeft);
SR_DeactivateLeftMeneu(SET1 := _rt18.Q, RESET := _rt19.Q); // SR
deactivateMainMeneu := SR_DeactivateLeftMeneu.Q1;
deactivateSeconderyMeneu := NOT SR_DeactivateLeftMeneu.Q1;

// NETWORK 27 (disabled)
// _rt20(CLK := GVL_KeyList.xRight);
// TON_Delay(IN := deactivateMainMeneu); // TON
// _rt21(CLK := GVL_KeyList.xLeft);
// SR_activate3rdColumn(SET1 := _rt20.Q AND TON_Delay.Q, RESET := _rt21.Q); // SR
// thirdColumnActive := SR_activate3rdColumn.Q1;

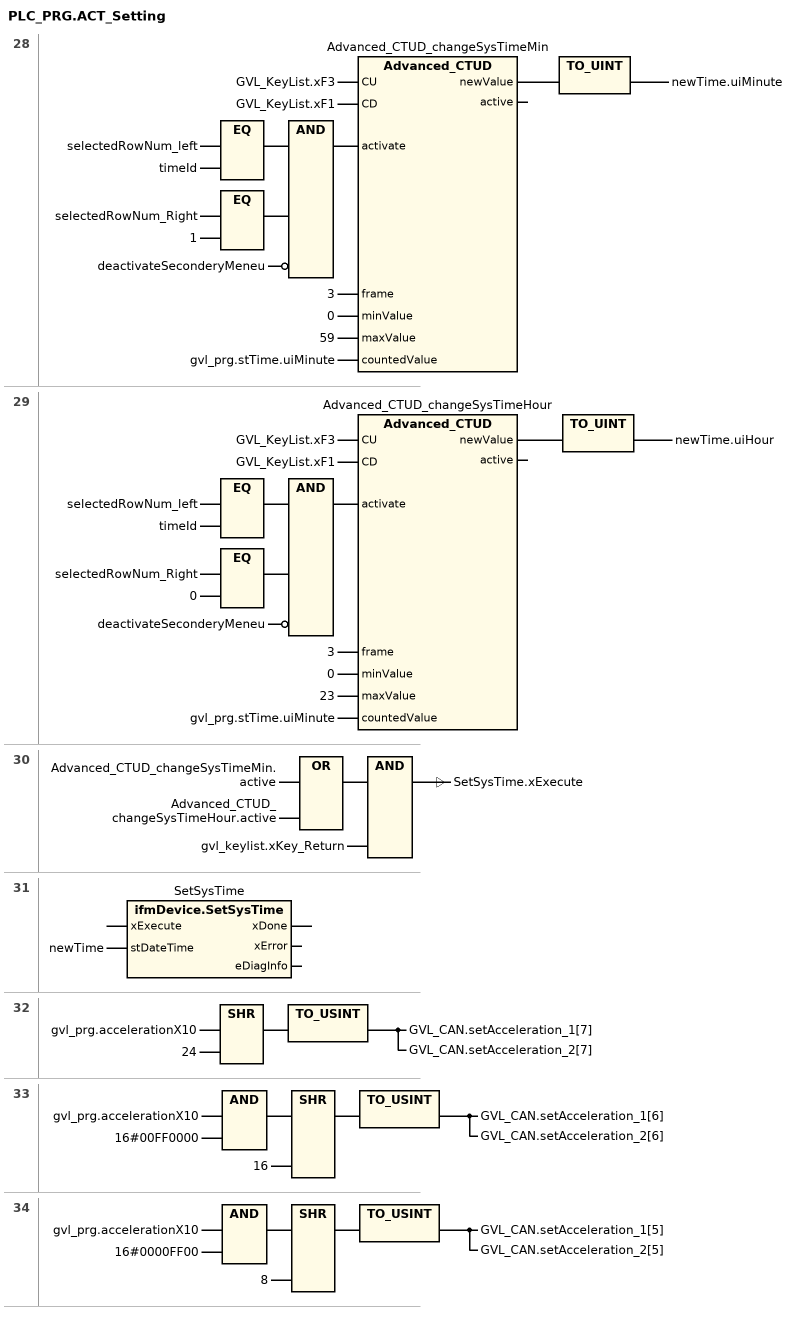
// NETWORK 28
Advanced_CTUD_changeSysTimeMin(
    CU := GVL_KeyList.xF3,
    CD := GVL_KeyList.xF1,
    activate := selectedRowNum_left = timeId AND selectedRowNum_Right = 1 AND NOT deactivateSeconderyMeneu,
    frame := 3,
    minValue := 0,
    maxValue := 59,
    countedValue := gvl_prg.stTime.uiMinute); // Advanced_CTUD
newTime.uiMinute := TO_UINT(Advanced_CTUD_changeSysTimeMin.newValue);

// NETWORK 29
Advanced_CTUD_changeSysTimeHour(
    CU := GVL_KeyList.xF3,
    CD := GVL_KeyList.xF1,
    activate := selectedRowNum_left = timeId AND selectedRowNum_Right = 0 AND NOT deactivateSeconderyMeneu,
    frame := 3,
    minValue := 0,
    maxValue := 23,
    countedValue := gvl_prg.stTime.uiMinute); // Advanced_CTUD
newTime.uiHour := TO_UINT(Advanced_CTUD_changeSysTimeHour.newValue);

// NETWORK 30
_rt22(CLK := (Advanced_CTUD_changeSysTimeMin.active OR Advanced_CTUD_changeSysTimeHour.active) AND gvl_keylist.xKey_Return);
SetSysTime.xExecute := _rt22.Q;

// NETWORK 31
SetSysTime(stDateTime := newTime); // ifmDevice.SetSysTime

// NETWORK 32
_w4 := TO_USINT(SHR(gvl_prg.accelerationX10, 24));
GVL_CAN.setAcceleration_1[7] := _w4;
GVL_CAN.setAcceleration_2[7] := _w4;

// NETWORK 33
_w5 := TO_USINT(SHR(gvl_prg.accelerationX10 AND 16#00FF0000, 16));
GVL_CAN.setAcceleration_1[6] := _w5;
GVL_CAN.setAcceleration_2[6] := _w5;

// NETWORK 34
_w6 := TO_USINT(SHR(gvl_prg.accelerationX10 AND 16#0000FF00, 8));
GVL_CAN.setAcceleration_1[5] := _w6;
GVL_CAN.setAcceleration_2[5] := _w6;

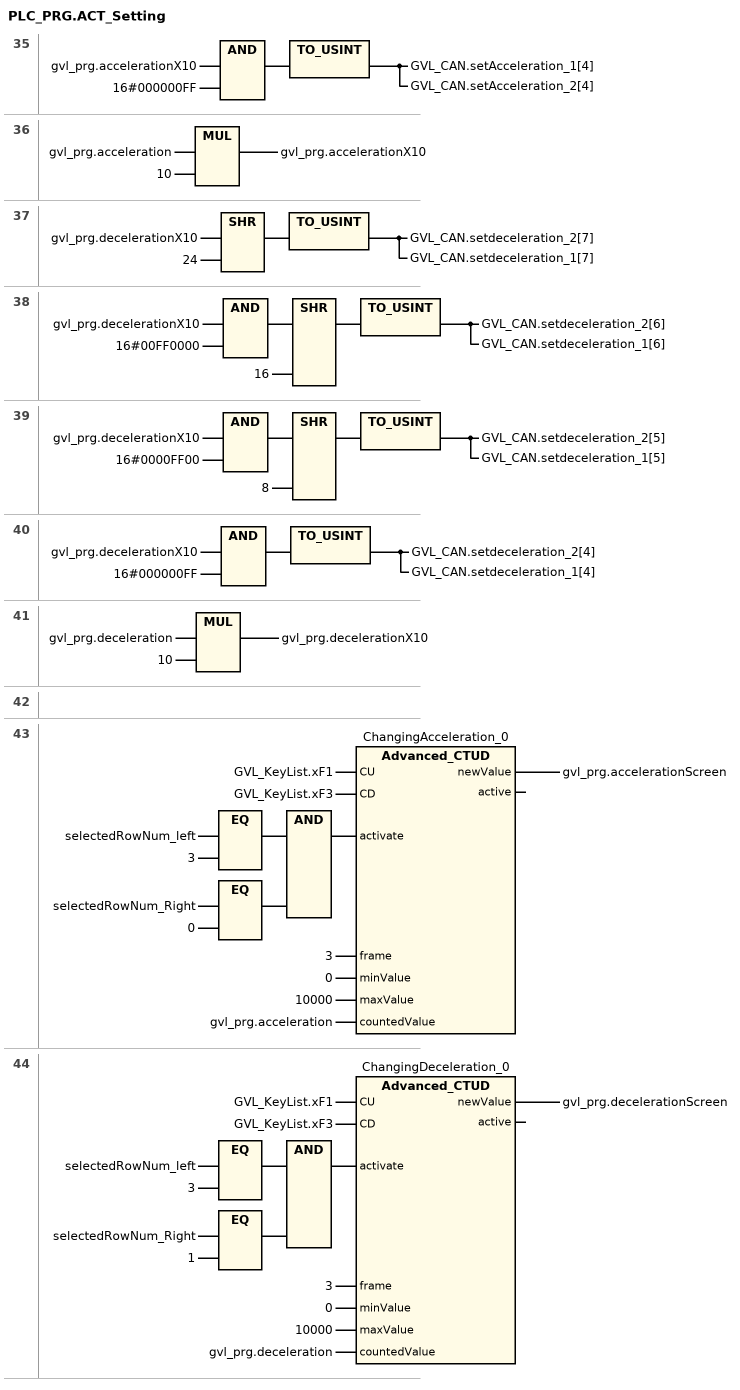
// NETWORK 35
_w7 := TO_USINT(gvl_prg.accelerationX10 AND 16#000000FF);
GVL_CAN.setAcceleration_1[4] := _w7;
GVL_CAN.setAcceleration_2[4] := _w7;

// NETWORK 36
gvl_prg.accelerationX10 := gvl_prg.acceleration * 10;

// NETWORK 37
_w8 := TO_USINT(SHR(gvl_prg.decelerationX10, 24));
GVL_CAN.setdeceleration_2[7] := _w8;
GVL_CAN.setdeceleration_1[7] := _w8;

// NETWORK 38
_w9 := TO_USINT(SHR(gvl_prg.decelerationX10 AND 16#00FF0000, 16));
GVL_CAN.setdeceleration_2[6] := _w9;
GVL_CAN.setdeceleration_1[6] := _w9;

// NETWORK 39
_w10 := TO_USINT(SHR(gvl_prg.decelerationX10 AND 16#0000FF00, 8));
GVL_CAN.setdeceleration_2[5] := _w10;
GVL_CAN.setdeceleration_1[5] := _w10;

// NETWORK 40
_w11 := TO_USINT(gvl_prg.decelerationX10 AND 16#000000FF);
GVL_CAN.setdeceleration_2[4] := _w11;
GVL_CAN.setdeceleration_1[4] := _w11;

// NETWORK 41
gvl_prg.decelerationX10 := gvl_prg.deceleration * 10;

// NETWORK 42

// NETWORK 43
ChangingAcceleration_0(
    CU := GVL_KeyList.xF1,
    CD := GVL_KeyList.xF3,
    activate := selectedRowNum_left = 3 AND selectedRowNum_Right = 0,
    frame := 3,
    minValue := 0,
    maxValue := 10000,
    countedValue := gvl_prg.acceleration); // Advanced_CTUD
gvl_prg.accelerationScreen := ChangingAcceleration_0.newValue;

// NETWORK 44
ChangingDeceleration_0(
    CU := GVL_KeyList.xF1,
    CD := GVL_KeyList.xF3,
    activate := selectedRowNum_left = 3 AND selectedRowNum_Right = 1,
    frame := 3,
    minValue := 0,
    maxValue := 10000,
    countedValue := gvl_prg.deceleration); // Advanced_CTUD
gvl_prg.decelerationScreen := ChangingDeceleration_0.newValue;

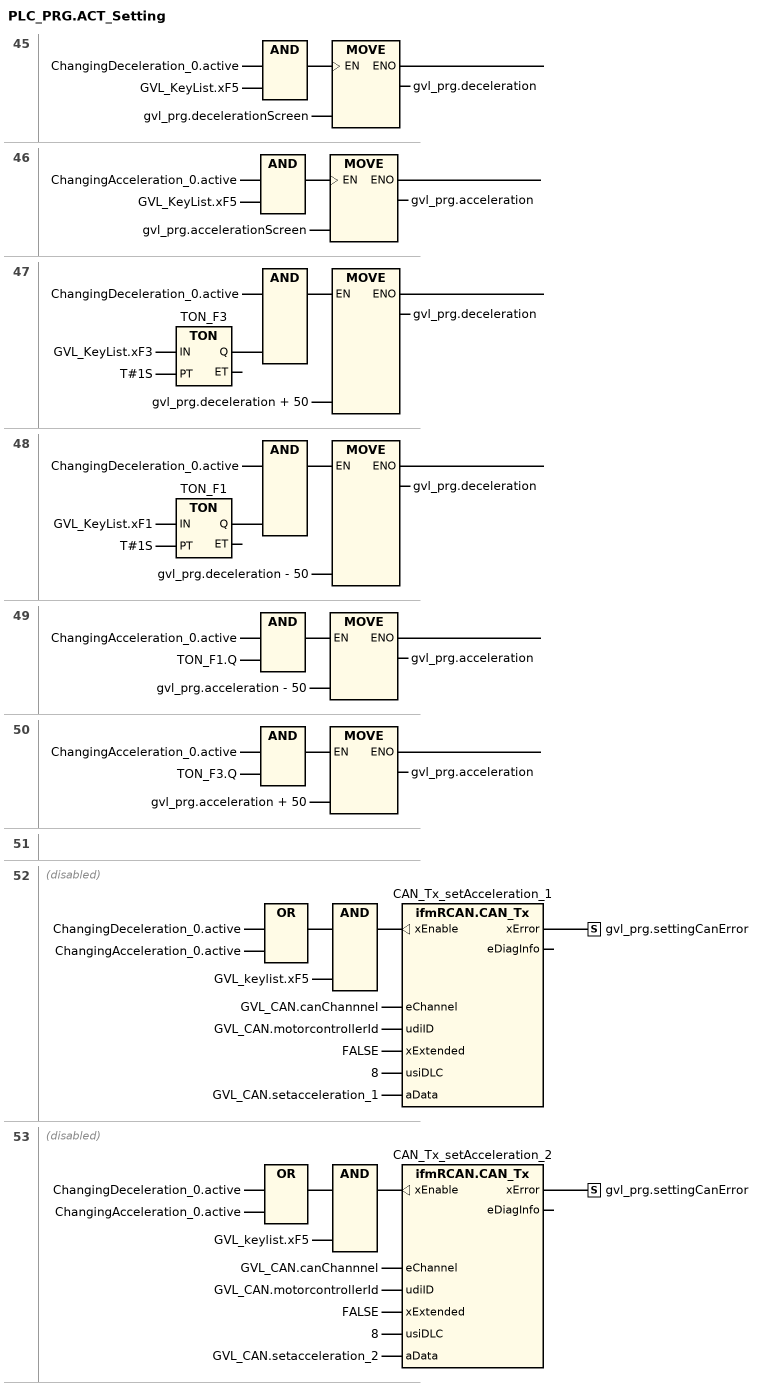
// NETWORK 45
_rt23(CLK := ChangingDeceleration_0.active AND GVL_KeyList.xF5);
IF _rt23.Q THEN gvl_prg.deceleration := gvl_prg.decelerationScreen; END_IF

// NETWORK 46
_rt24(CLK := ChangingAcceleration_0.active AND GVL_KeyList.xF5);
IF _rt24.Q THEN gvl_prg.acceleration := gvl_prg.accelerationScreen; END_IF

// NETWORK 47
TON_F3(IN := GVL_KeyList.xF3, PT := T#1S); // TON
IF ChangingDeceleration_0.active AND TON_F3.Q THEN gvl_prg.deceleration := gvl_prg.deceleration + 50; END_IF

// NETWORK 48
TON_F1(IN := GVL_KeyList.xF1, PT := T#1S); // TON
IF ChangingDeceleration_0.active AND TON_F1.Q THEN gvl_prg.deceleration := gvl_prg.deceleration - 50; END_IF

// NETWORK 49
IF ChangingAcceleration_0.active AND TON_F1.Q THEN gvl_prg.acceleration := gvl_prg.acceleration - 50; END_IF

// NETWORK 50
IF ChangingAcceleration_0.active AND TON_F3.Q THEN gvl_prg.acceleration := gvl_prg.acceleration + 50; END_IF

// NETWORK 51

// NETWORK 52 (disabled)
// _ft5(CLK := (ChangingDeceleration_0.active OR ChangingAcceleration_0.active) AND GVL_keylist.xF5);
// CAN_Tx_setAcceleration_1(
//     xEnable := _ft5.Q,
//     eChannel := GVL_CAN.canChannnel,
//     udiID := GVL_CAN.motorcontrollerId,
//     xExtended := FALSE,
//     usiDLC := 8,
//     aData := GVL_CAN.setacceleration_1); // ifmRCAN.CAN_Tx
// gvl_prg.settingCanError S= CAN_Tx_setAcceleration_1.xError;

// NETWORK 53 (disabled)
// _ft6(CLK := (ChangingDeceleration_0.active OR ChangingAcceleration_0.active) AND GVL_keylist.xF5);
// CAN_Tx_setAcceleration_2(
//     xEnable := _ft6.Q,
//     eChannel := GVL_CAN.canChannnel,
//     udiID := GVL_CAN.motorcontrollerId,
//     xExtended := FALSE,
//     usiDLC := 8,
//     aData := GVL_CAN.setacceleration_2); // ifmRCAN.CAN_Tx
// gvl_prg.settingCanError S= CAN_Tx_setAcceleration_2.xError;

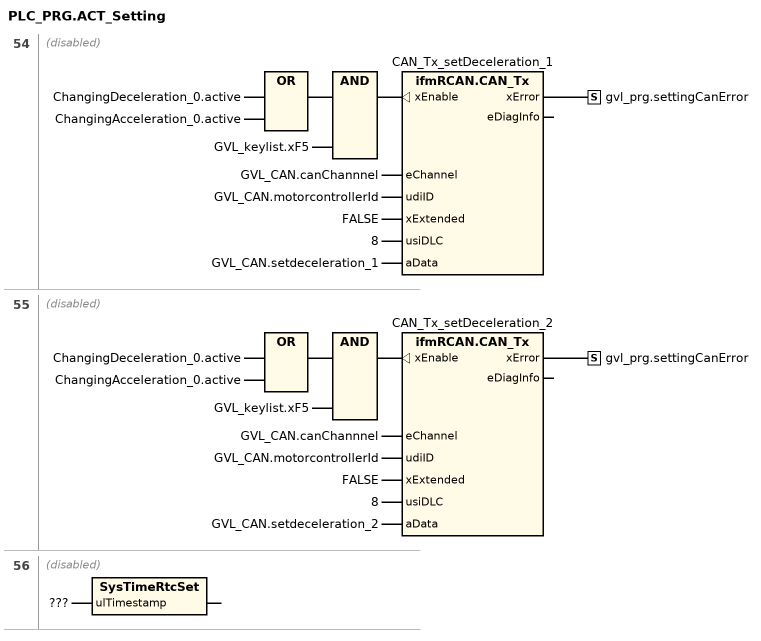
// NETWORK 54 (disabled)
// _ft7(CLK := (ChangingDeceleration_0.active OR ChangingAcceleration_0.active) AND GVL_keylist.xF5);
// CAN_Tx_setDeceleration_1(
//     xEnable := _ft7.Q,
//     eChannel := GVL_CAN.canChannnel,
//     udiID := GVL_CAN.motorcontrollerId,
//     xExtended := FALSE,
//     usiDLC := 8,
//     aData := GVL_CAN.setdeceleration_1); // ifmRCAN.CAN_Tx
// gvl_prg.settingCanError S= CAN_Tx_setDeceleration_1.xError;

// NETWORK 55 (disabled)
// _ft8(CLK := (ChangingDeceleration_0.active OR ChangingAcceleration_0.active) AND GVL_keylist.xF5);
// CAN_Tx_setDeceleration_2(
//     xEnable := _ft8.Q,
//     eChannel := GVL_CAN.canChannnel,
//     udiID := GVL_CAN.motorcontrollerId,
//     xExtended := FALSE,
//     usiDLC := 8,
//     aData := GVL_CAN.setdeceleration_2); // ifmRCAN.CAN_Tx
// gvl_prg.settingCanError S= CAN_Tx_setDeceleration_2.xError;

// NETWORK 56 (disabled)
// SysTimeRtcSet();
END_ACTION

ACTION ACT_PressedKeysConfig:
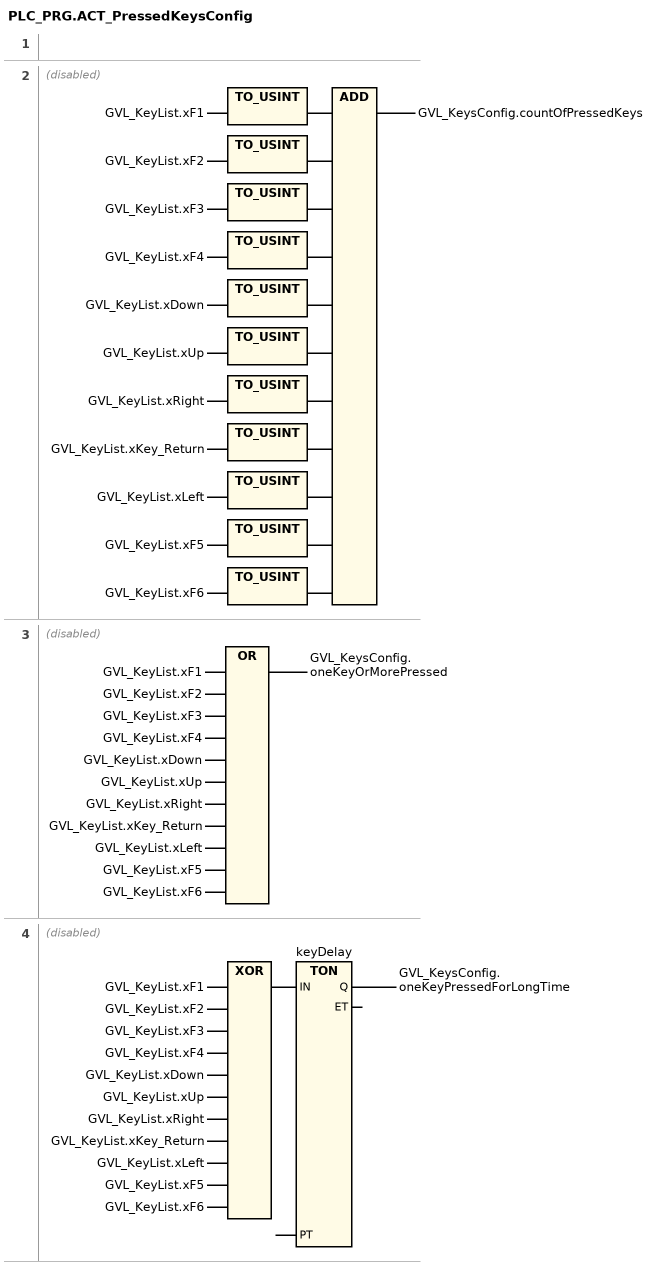
// NETWORK 1

// NETWORK 2 (disabled)
// GVL_KeysConfig.countOfPressedKeys := TO_USINT(GVL_KeyList.xF1) + TO_USINT(GVL_KeyList.xF2) + TO_USINT(GVL_KeyList.xF3) + TO_USINT(GVL_KeyList.xF4) + TO_USINT(GVL_KeyList.xDown) + TO_USINT(GVL_KeyList.xUp) + TO_USINT(GVL_KeyList.xRight) + TO_USINT(GVL_KeyList.xKey_Return) + TO_USINT(GVL_KeyList.xLeft) + TO_USINT(GVL_KeyList.xF5) + TO_USINT(GVL_KeyList.xF6);

// NETWORK 3 (disabled)
// GVL_KeysConfig.oneKeyOrMorePressed := GVL_KeyList.xF1 OR GVL_KeyList.xF2 OR GVL_KeyList.xF3 OR GVL_KeyList.xF4 OR GVL_KeyList.xDown OR GVL_KeyList.xUp OR GVL_KeyList.xRight OR GVL_KeyList.xKey_Return OR GVL_KeyList.xLeft OR GVL_KeyList.xF5 OR GVL_KeyList.xF6;

// NETWORK 4 (disabled)
// keyDelay(IN := GVL_KeyList.xF1 XOR GVL_KeyList.xF2 XOR GVL_KeyList.xF3 XOR GVL_KeyList.xF4 XOR GVL_KeyList.xDown XOR GVL_KeyList.xUp XOR GVL_KeyList.xRight XOR GVL_KeyList.xKey_Return XOR GVL_KeyList.xLeft XOR GVL_KeyList.xF5 XOR GVL_KeyList.xF6); // TON
// GVL_KeysConfig.oneKeyPressedForLongTime := keyDelay.Q;
END_ACTION

ACTION ACT_Button_Control:
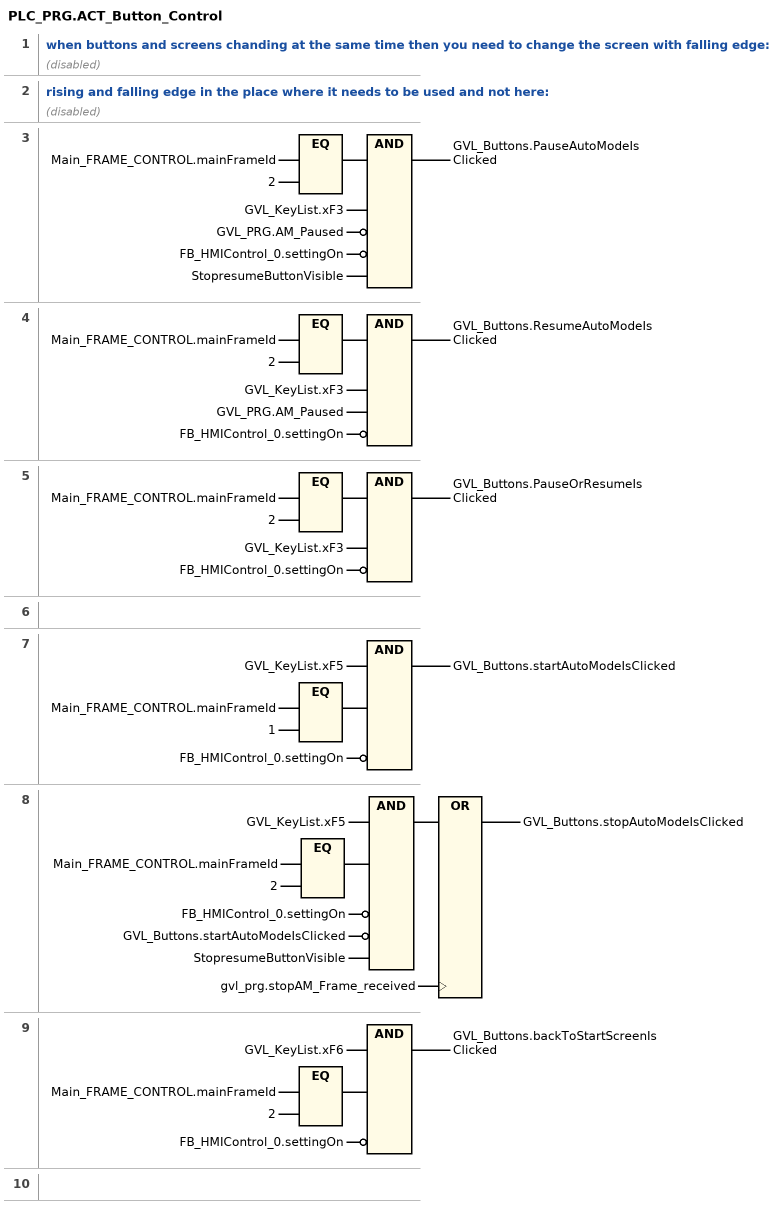
// NETWORK 1 (disabled)
// label: when buttons and screens chanding at the same time then you need to change the screen with falling edge

// NETWORK 2 (disabled)
// label: rising and falling edge in the place where it needs to be used and not here

// NETWORK 3
GVL_Buttons.PauseAutoModeIsClicked := Main_FRAME_CONTROL.mainFrameId = 2 AND GVL_KeyList.xF3 AND NOT GVL_PRG.AM_Paused AND NOT FB_HMIControl_0.settingOn AND StopresumeButtonVisible;

// NETWORK 4
GVL_Buttons.ResumeAutoModeIsClicked := Main_FRAME_CONTROL.mainFrameId = 2 AND GVL_KeyList.xF3 AND GVL_PRG.AM_Paused AND NOT FB_HMIControl_0.settingOn;

// NETWORK 5
GVL_Buttons.PauseOrResumeIsClicked := Main_FRAME_CONTROL.mainFrameId = 2 AND GVL_KeyList.xF3 AND NOT FB_HMIControl_0.settingOn;

// NETWORK 6

// NETWORK 7
GVL_Buttons.startAutoModeIsClicked := GVL_KeyList.xF5 AND Main_FRAME_CONTROL.mainFrameId = 1 AND NOT FB_HMIControl_0.settingOn;

// NETWORK 8
_rt25(CLK := gvl_prg.stopAM_Frame_received);
GVL_Buttons.stopAutoModeIsClicked := GVL_KeyList.xF5 AND Main_FRAME_CONTROL.mainFrameId = 2 AND NOT FB_HMIControl_0.settingOn AND NOT GVL_Buttons.startAutoModeIsClicked AND StopresumeButtonVisible OR _rt25.Q;

// NETWORK 9
GVL_Buttons.backToStartScreenIsClicked := GVL_KeyList.xF6 AND Main_FRAME_CONTROL.mainFrameId = 2 AND NOT FB_HMIControl_0.settingOn;

// NETWORK 10

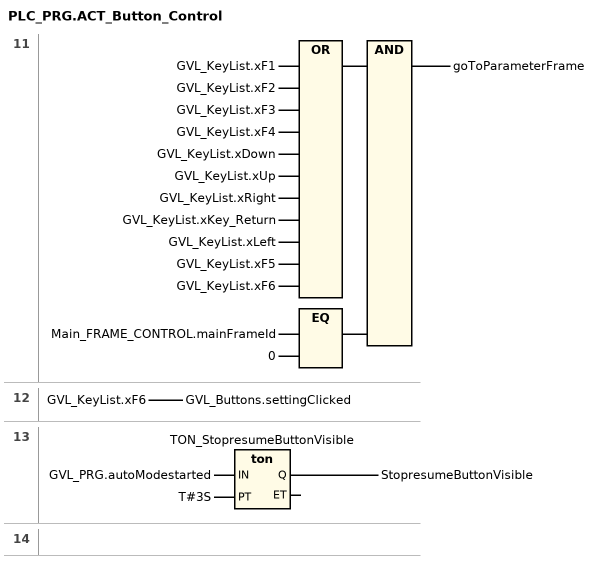
// NETWORK 11
goToParameterFrame := (GVL_KeyList.xF1 OR GVL_KeyList.xF2 OR GVL_KeyList.xF3 OR GVL_KeyList.xF4 OR GVL_KeyList.xDown OR GVL_KeyList.xUp OR GVL_KeyList.xRight OR GVL_KeyList.xKey_Return OR GVL_KeyList.xLeft OR GVL_KeyList.xF5 OR GVL_KeyList.xF6) AND Main_FRAME_CONTROL.mainFrameId = 0;

// NETWORK 12
GVL_Buttons.settingClicked := GVL_KeyList.xF6;

// NETWORK 13
TON_StopresumeButtonVisible(IN := GVL_PRG.autoModestarted, PT := T#3S); // ton
StopresumeButtonVisible := TON_StopresumeButtonVisible.Q;

// NETWORK 14
END_ACTION

END_PROGRAM

// Device/Application/FBs/changeLanguage
FUNCTION_BLOCK changeLanguage
VAR_INPUT
	stLaunguage: STRING := 'DE';
END_VAR
VAR_OUTPUT
END_VAR
VAR
END_VAR

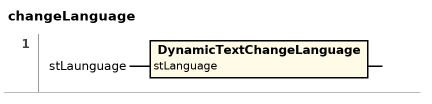
// NETWORK 1
DynamicTextChangeLanguage(stLanguage := stLaunguage);

END_FUNCTION_BLOCK

// Device/Application/FBs/Controll/HMIControl
FUNCTION_BLOCK HMIControl
VAR_INPUT
	//nextRow:BOOL;
	bDirection: BOOL;
	countOfRows: USINT;
	
END_VAR
VAR_OUTPUT
	selectedParameterIndex: USINT;
	editRowParameterEn: BOOL;
	stTime : ifmDevice.stDATE_TIME; // system time
	settingOn : BOOL;
END_VAR
VAR

	ControlAllKeyLEDs_0: ifmDevice.SetKeyLED;
	SetStatusLEDstate_0: ifmDevice.SetStatusLEDstate;
	GetSysResources_0: ifmDevice.GetSysResources;
	CAN_Enable_0: ifmRCAN.CAN_Enable;
	coreUsage0: USINT:= 0;
	coreUsage1:  USINT:= 0;
	
	// locationsite
	goToLocationSite: BOOL;
	//switschingToAutoModeSite: BOOL;
	//help1 : BOOL;
	//buttonsControl_0: ButtonControl;

	GetSysTime_0: ifmDevice.GetSysTime;
	
	RS_get_Time: Standard.RS;
	TON_timeUpdatefreq: Standard.TON;
	eDialogDone :ifmTypes2.eDIAG_INFO  := ifmTypes2.eDIAG_INFO.STAT_DONE;
	RS_settingOn: Standard.RS ;

	CTUD_StartMin: CTUD;
	SR_editingStartTimeActive: SR;
	RS_StartTimeEdited: RS;
	CTUD_StartHour: CTUD;
	sttedStartTime: STRING(255);
	FB_smoothCLK_starttimeHourCD: FB_smoothCLK;
	FB_smoothCLK_starttimeHourCU: FB_smoothCLK;
	FB_smoothCLK_starttimeMinCD: FB_smoothCLK;
	FB_smoothCLK_starttimeMinCU: FB_smoothCLK;
	ChangingStartTimeMin: Advanced_CTUD;
	FB_CLK_0: FB_CLK;
	test: UINT (0..23);
	test2: UINT (0..59);
	clk1: FB_CLK;
	
	shownStartTimeMin: INT;
	shownStartTimeHour: INT;
	ChangingStartTimeHour: Advanced_CTUD;
	helpVar2: INT;
	helpVar1: INT;
	SR_showKeys: sr;
	TON_ShowKeys: ton;
	RS_get_Time1: RS;
	LoadSplashScreen_0: ifmDevice.LoadSplashScreen;
	TON_hideKeys : TON;

END_VAR
VAR // added by the converter: edge detectors and wires of the graphical bodies
    _rt1, _rt2, _rt3, _rt4, _rt5, _rt6, _rt7, _rt8, _rt9, _rt10 : R_TRIG;
    _w1, _w2 : BOOL;
    _ft1 : F_TRIG;
END_VAR

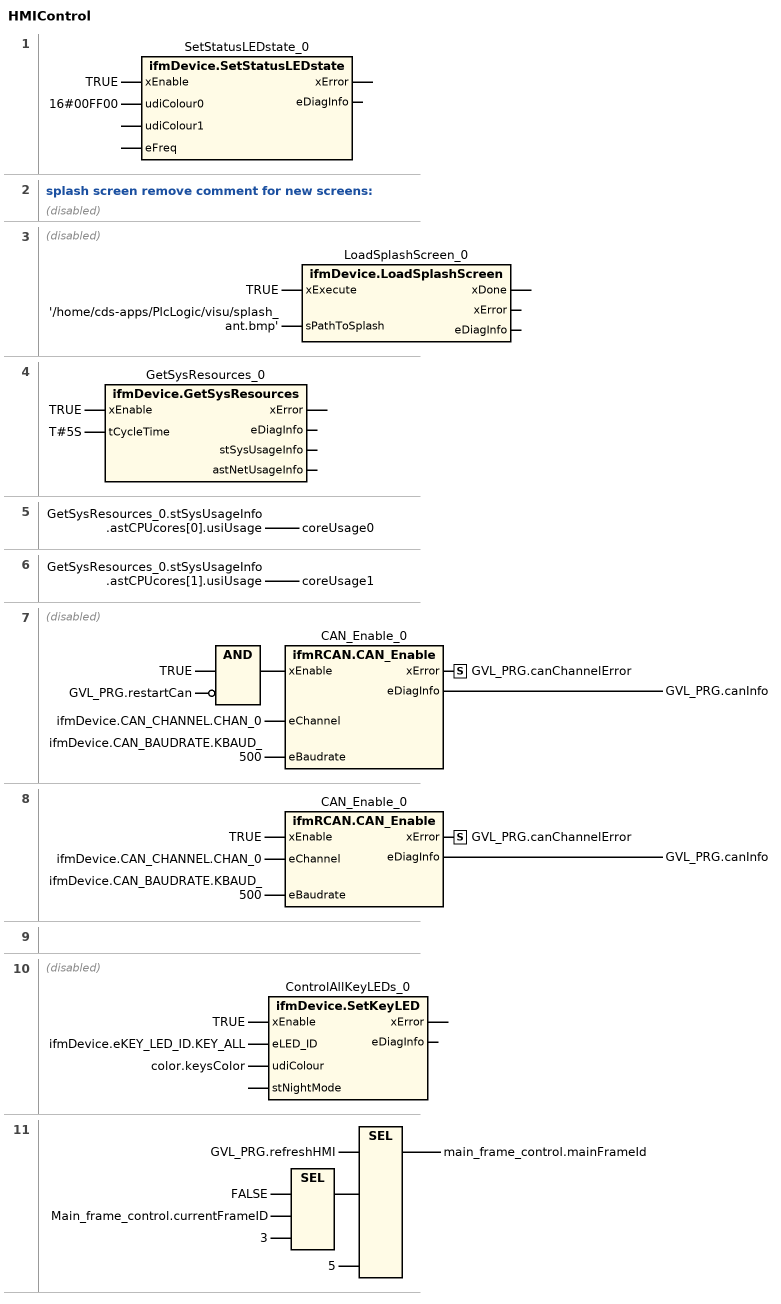
// NETWORK 1
SetStatusLEDstate_0(xEnable := TRUE, udiColour0 := 16#00FF00); // ifmDevice.SetStatusLEDstate

// NETWORK 2 (disabled)
// label: splash screen remove comment for new screens

// NETWORK 3 (disabled)
// LoadSplashScreen_0(xExecute := TRUE, sPathToSplash := '/home/cds-apps/PlcLogic/visu/splash_ant.bmp'); // ifmDevice.LoadSplashScreen

// NETWORK 4
GetSysResources_0(xEnable := TRUE, tCycleTime := T#5S); // ifmDevice.GetSysResources

// NETWORK 5
coreUsage0 := GetSysResources_0.stSysUsageInfo .astCPUcores[0].usiUsage;

// NETWORK 6
coreUsage1 := GetSysResources_0.stSysUsageInfo .astCPUcores[1].usiUsage;

// NETWORK 7 (disabled)
// CAN_Enable_0(
//     xEnable := TRUE AND NOT GVL_PRG.restartCan,
//     eChannel := ifmDevice.CAN_CHANNEL.CHAN_0,
//     eBaudrate := ifmDevice.CAN_BAUDRATE.KBAUD_500); // ifmRCAN.CAN_Enable
// GVL_PRG.canChannelError S= CAN_Enable_0.xError;
// GVL_PRG.canInfo := CAN_Enable_0.eDiagInfo;

// NETWORK 8
CAN_Enable_0(
    xEnable := TRUE,
    eChannel := ifmDevice.CAN_CHANNEL.CHAN_0,
    eBaudrate := ifmDevice.CAN_BAUDRATE.KBAUD_500); // ifmRCAN.CAN_Enable
GVL_PRG.canChannelError S= CAN_Enable_0.xError;
GVL_PRG.canInfo := CAN_Enable_0.eDiagInfo;

// NETWORK 9

// NETWORK 10 (disabled)
// ControlAllKeyLEDs_0(xEnable := TRUE, eLED_ID := ifmDevice.eKEY_LED_ID.KEY_ALL, udiColour := color.keysColor); // ifmDevice.SetKeyLED

// NETWORK 11
main_frame_control.mainFrameId := SEL(GVL_PRG.refreshHMI, SEL(FALSE, Main_frame_control.currentFrameID, 3), 5);

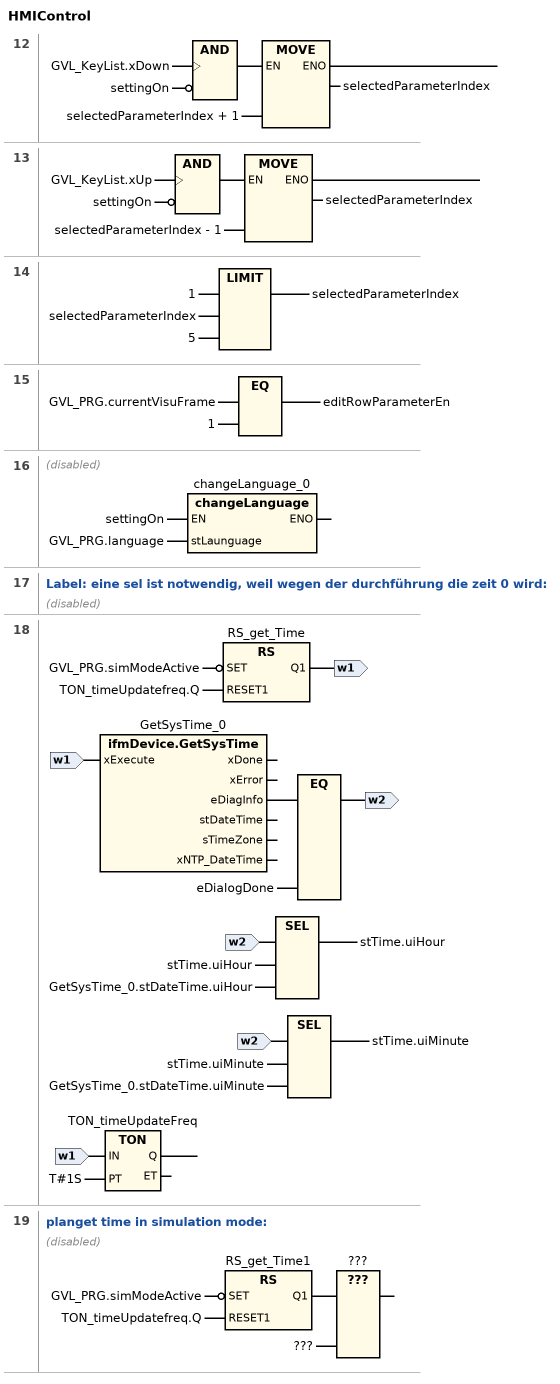
// NETWORK 12
_rt1(CLK := GVL_KeyList.xDown);
IF _rt1.Q AND NOT settingOn THEN selectedParameterIndex := selectedParameterIndex + 1; END_IF

// NETWORK 13
_rt2(CLK := GVL_KeyList.xUp);
IF _rt2.Q AND NOT settingOn THEN selectedParameterIndex := selectedParameterIndex - 1; END_IF

// NETWORK 14
selectedParameterIndex := LIMIT(1, selectedParameterIndex, 5);

// NETWORK 15
editRowParameterEn := GVL_PRG.currentVisuFrame = 1;

// NETWORK 16 (disabled)
// IF settingOn THEN
//     changeLanguage_0(stLaunguage := GVL_PRG.language); // changeLanguage
// END_IF

// NETWORK 17 (disabled)
// label: Label: eine sel ist notwendig, weil wegen der durchführung die zeit 0 wird

// NETWORK 18
RS_get_Time(SET := NOT GVL_PRG.simModeActive, RESET1 := TON_timeUpdatefreq.Q); // RS
GetSysTime_0(xExecute := RS_get_Time.Q1); // ifmDevice.GetSysTime
_w1 := GetSysTime_0.eDiagInfo = eDialogDone;
stTime.uiHour := SEL(_w1, stTime.uiHour, GetSysTime_0.stDateTime.uiHour);
stTime.uiMinute := SEL(_w1, stTime.uiMinute, GetSysTime_0.stDateTime.uiMinute);
TON_timeUpdateFreq(IN := RS_get_Time.Q1, PT := T#1S); // TON

// NETWORK 19 (disabled)
// label: planget time in simulation mode
// RS_get_Time1(SET := NOT GVL_PRG.simModeActive, RESET1 := TON_timeUpdatefreq.Q); // RS
// ???(IN1 := RS_get_Time1.Q1);

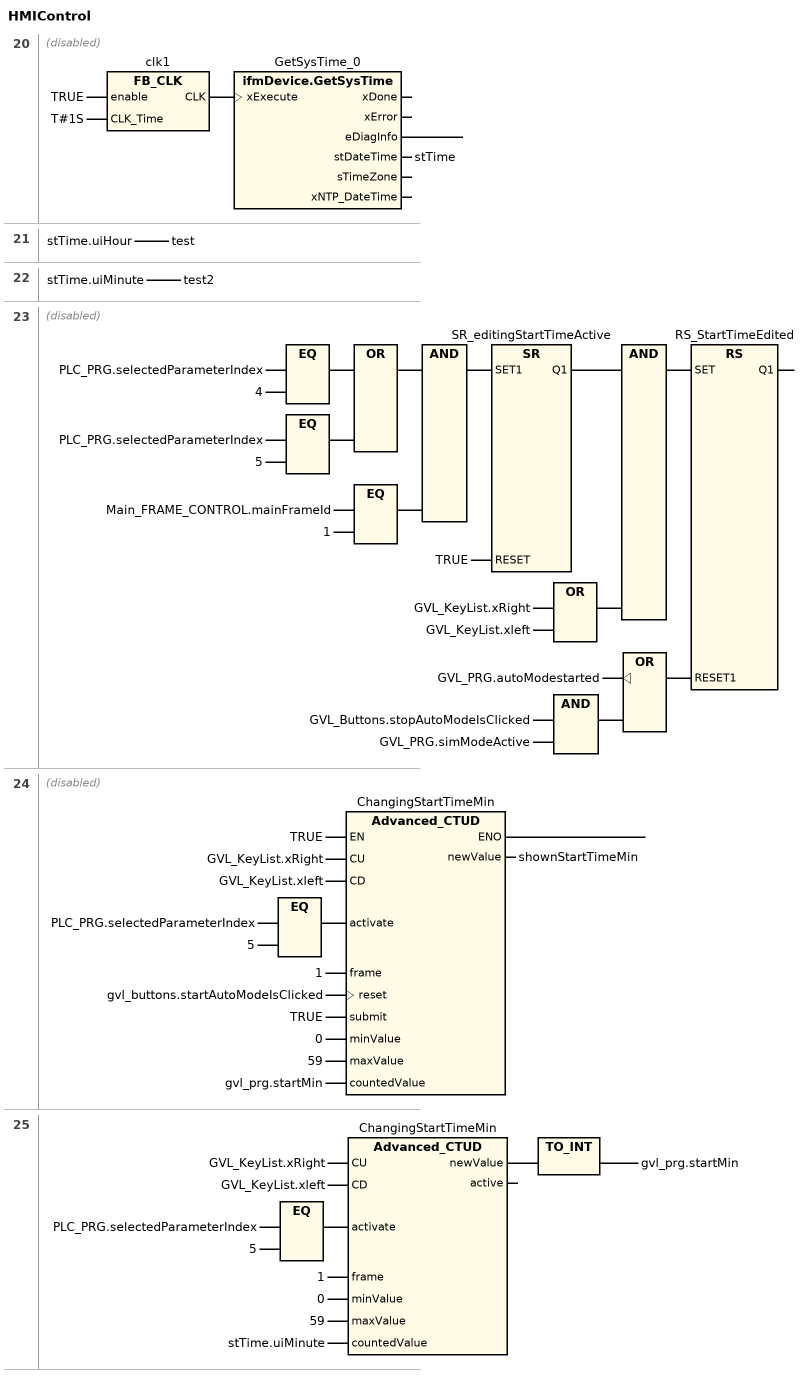
// NETWORK 20 (disabled)
// clk1(enable := TRUE, CLK_Time := T#1S); // FB_CLK
// _rt3(CLK := clk1.CLK);
// GetSysTime_0(xExecute := _rt3.Q, stDateTime => stTime); // ifmDevice.GetSysTime

// NETWORK 21
test := stTime.uiHour;

// NETWORK 22
test2 := stTime.uiMinute;

// NETWORK 23 (disabled)
// SR_editingStartTimeActive(SET1 := (PLC_PRG.selectedParameterIndex = 4 OR PLC_PRG.selectedParameterIndex = 5) AND Main_FRAME_CONTROL.mainFrameId = 1, RESET := TRUE); // SR
// _ft1(CLK := GVL_PRG.autoModestarted);
// RS_StartTimeEdited(SET := SR_editingStartTimeActive.Q1 AND (GVL_KeyList.xRight OR GVL_KeyList.xleft), RESET1 := _ft1.Q OR GVL_Buttons.stopAutoModeIsClicked AND GVL_PRG.simModeActive); // RS

// NETWORK 24 (disabled)
// _rt4(CLK := gvl_buttons.startAutoModeIsClicked);
// ChangingStartTimeMin(
//     CU := GVL_KeyList.xRight,
//     CD := GVL_KeyList.xleft,
//     activate := PLC_PRG.selectedParameterIndex = 5,
//     frame := 1,
//     reset := _rt4.Q,
//     submit := TRUE,
//     minValue := 0,
//     maxValue := 59,
//     countedValue := gvl_prg.startMin,
//     newValue => shownStartTimeMin); // Advanced_CTUD

// NETWORK 25
ChangingStartTimeMin(
    CU := GVL_KeyList.xRight,
    CD := GVL_KeyList.xleft,
    activate := PLC_PRG.selectedParameterIndex = 5,
    frame := 1,
    minValue := 0,
    maxValue := 59,
    countedValue := stTime.uiMinute); // Advanced_CTUD
gvl_prg.startMin := TO_INT(ChangingStartTimeMin.newValue);

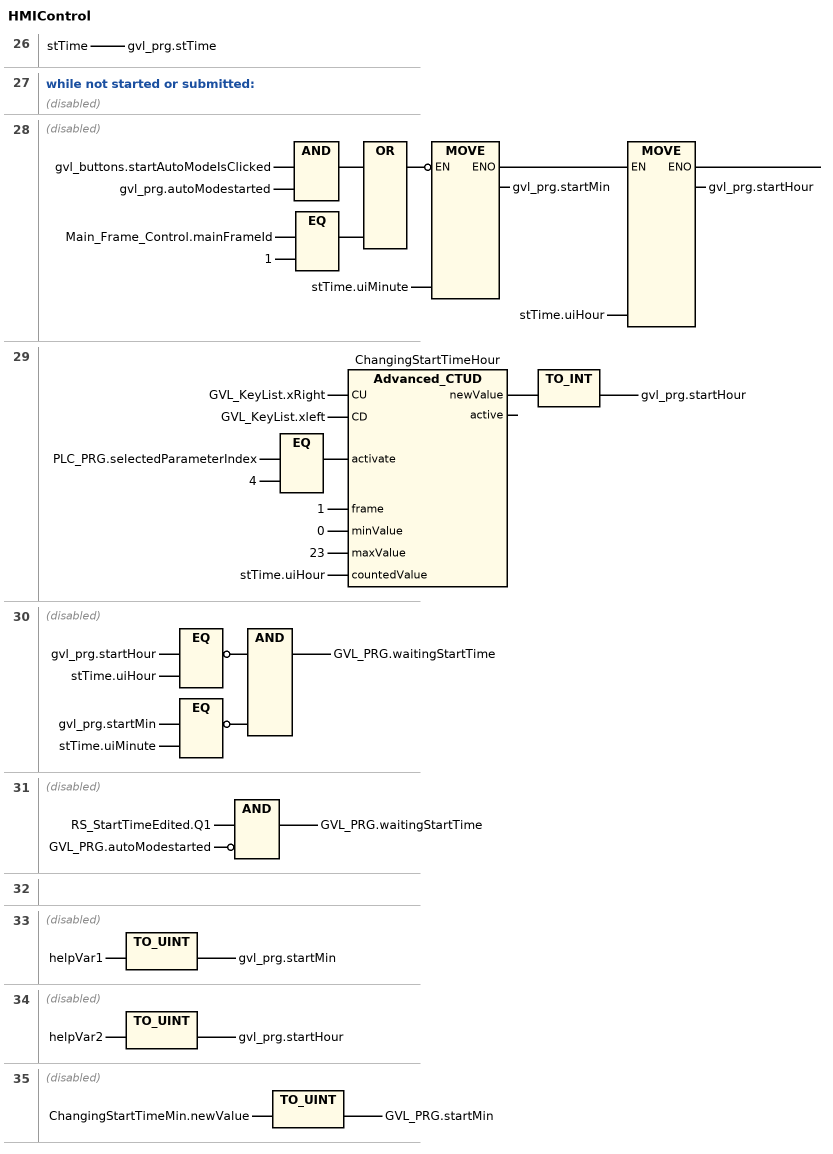
// NETWORK 26
gvl_prg.stTime := stTime;

// NETWORK 27 (disabled)
// label: while not started or submitted

// NETWORK 28 (disabled)
// _w2 := NOT (gvl_buttons.startAutoModeIsClicked AND gvl_prg.autoModestarted OR Main_Frame_Control.mainFrameId = 1);
// IF _w2 THEN gvl_prg.startMin := stTime.uiMinute; END_IF
// IF _w2 THEN gvl_prg.startHour := stTime.uiHour; END_IF

// NETWORK 29
ChangingStartTimeHour(
    CU := GVL_KeyList.xRight,
    CD := GVL_KeyList.xleft,
    activate := PLC_PRG.selectedParameterIndex = 4,
    frame := 1,
    minValue := 0,
    maxValue := 23,
    countedValue := stTime.uiHour); // Advanced_CTUD
gvl_prg.startHour := TO_INT(ChangingStartTimeHour.newValue);

// NETWORK 30 (disabled)
// GVL_PRG.waitingStartTime := NOT (gvl_prg.startHour = stTime.uiHour) AND NOT (gvl_prg.startMin = stTime.uiMinute);

// NETWORK 31 (disabled)
// GVL_PRG.waitingStartTime := RS_StartTimeEdited.Q1 AND NOT GVL_PRG.autoModestarted;

// NETWORK 32

// NETWORK 33 (disabled)
// gvl_prg.startMin := TO_UINT(helpVar1);

// NETWORK 34 (disabled)
// gvl_prg.startHour := TO_UINT(helpVar2);

// NETWORK 35 (disabled)
// GVL_PRG.startMin := TO_UINT(ChangingStartTimeMin.newValue);

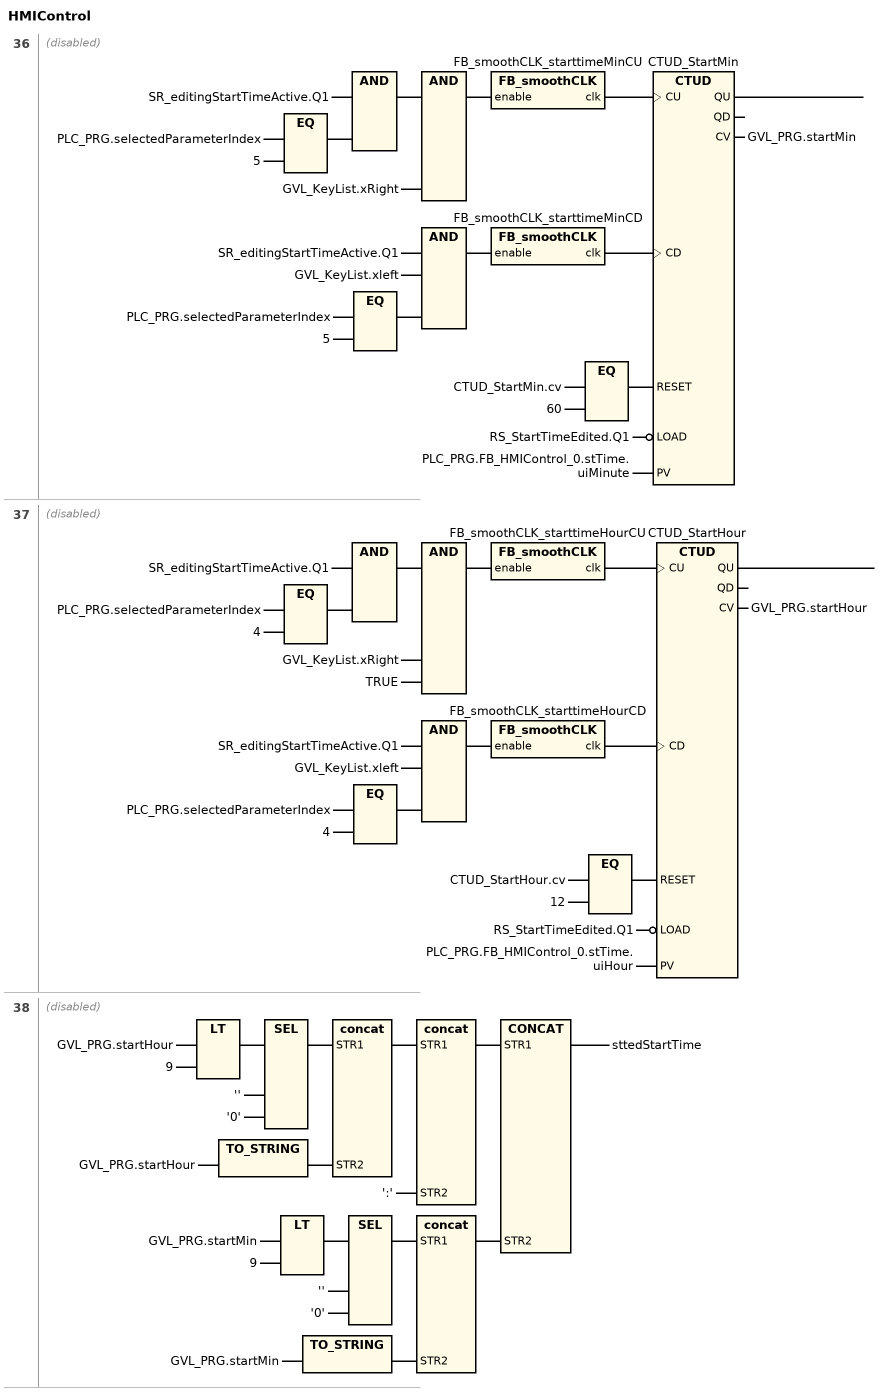
// NETWORK 36 (disabled)
// FB_smoothCLK_starttimeMinCU(enable := (SR_editingStartTimeActive.Q1 AND PLC_PRG.selectedParameterIndex = 5) AND GVL_KeyList.xRight); // FB_smoothCLK
// _rt5(CLK := FB_smoothCLK_starttimeMinCU.clk);
// FB_smoothCLK_starttimeMinCD(enable := SR_editingStartTimeActive.Q1 AND GVL_KeyList.xleft AND PLC_PRG.selectedParameterIndex = 5); // FB_smoothCLK
// _rt6(CLK := FB_smoothCLK_starttimeMinCD.clk);
// CTUD_StartMin(
//     CU := _rt5.Q,
//     CD := _rt6.Q,
//     RESET := CTUD_StartMin.cv = 60,
//     LOAD := NOT RS_StartTimeEdited.Q1,
//     PV := PLC_PRG.FB_HMIControl_0.stTime.uiMinute,
//     CV => GVL_PRG.startMin); // CTUD

// NETWORK 37 (disabled)
// FB_smoothCLK_starttimeHourCU(enable := (SR_editingStartTimeActive.Q1 AND PLC_PRG.selectedParameterIndex = 4) AND GVL_KeyList.xRight AND TRUE); // FB_smoothCLK
// _rt7(CLK := FB_smoothCLK_starttimeHourCU.clk);
// FB_smoothCLK_starttimeHourCD(enable := SR_editingStartTimeActive.Q1 AND GVL_KeyList.xleft AND PLC_PRG.selectedParameterIndex = 4); // FB_smoothCLK
// _rt8(CLK := FB_smoothCLK_starttimeHourCD.clk);
// CTUD_StartHour(
//     CU := _rt7.Q,
//     CD := _rt8.Q,
//     RESET := CTUD_StartHour.cv = 12,
//     LOAD := NOT RS_StartTimeEdited.Q1,
//     PV := PLC_PRG.FB_HMIControl_0.stTime.uiHour,
//     CV => GVL_PRG.startHour); // CTUD

// NETWORK 38 (disabled)
// sttedStartTime := CONCAT(STR1 := concat(STR1 := concat(STR1 := SEL(GVL_PRG.startHour < 9, '', '0'), STR2 := TO_STRING(GVL_PRG.startHour)), STR2 := ':'), STR2 := concat(STR1 := SEL(GVL_PRG.startMin < 9, '', '0'), STR2 := TO_STRING(GVL_PRG.startMin)));

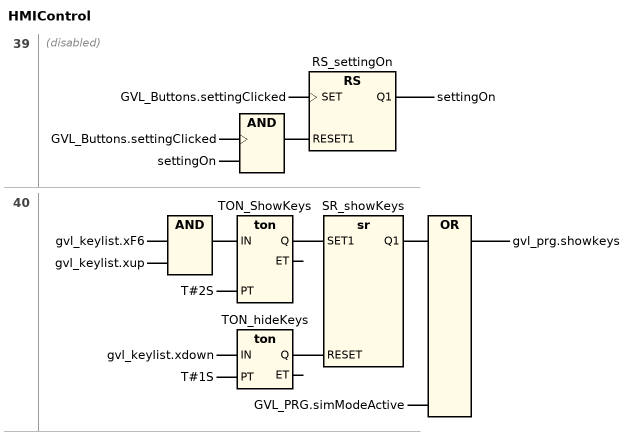
// NETWORK 39 (disabled)
// _rt9(CLK := GVL_Buttons.settingClicked);
// _rt10(CLK := GVL_Buttons.settingClicked);
// RS_settingOn(SET := _rt9.Q, RESET1 := _rt10.Q AND settingOn); // RS
// settingOn := RS_settingOn.Q1;

// NETWORK 40
TON_ShowKeys(IN := gvl_keylist.xF6 AND gvl_keylist.xup, PT := T#2S); // ton
TON_hideKeys(IN := gvl_keylist.xdown, PT := T#1S); // ton
SR_showKeys(SET1 := TON_ShowKeys.Q, RESET := TON_hideKeys.Q); // sr
gvl_prg.showkeys := SR_showKeys.Q1 OR GVL_PRG.simModeActive;

END_FUNCTION_BLOCK

// Device/Application/Programms/Main_FRAME_CONTROL
PROGRAM Main_FRAME_CONTROL
VAR_INPUT
		mainFrameId : USINT;
END_VAR
VAR
	currentFrameID :USINT;

	Delay : TON := (PT:= T#500MS);
	RS_Delay : RS;
	hv1: BOOL;
	RS_refreshHmi: RS;
	TON_refreshDelay: TON;
	TON_delay1: TON;
	TON_delay2: TON;
	RS_refreshCyclic: RS;
	TON_refreshCycleTime : TON := (PT := T#10S);
	TON_delay3: TON;
	SR_startFrame: sr;
	FB_CLK_0: fb_clk;
	cyclicRefresh: BOOL:= TRUE;
	fb_reduceActiveTime: fb_delay;
END_VAR
VAR // added by the converter: edge detectors and wires of the graphical bodies
    _rt1, _rt2, _rt3, _rt4 : R_TRIG;
    _ft1, _ft2, _ft3, _ft4, _ft5 : F_TRIG;
    _w1, _w2, _w3, _w4, _w5, _w6, _w7 : BOOL;
END_VAR

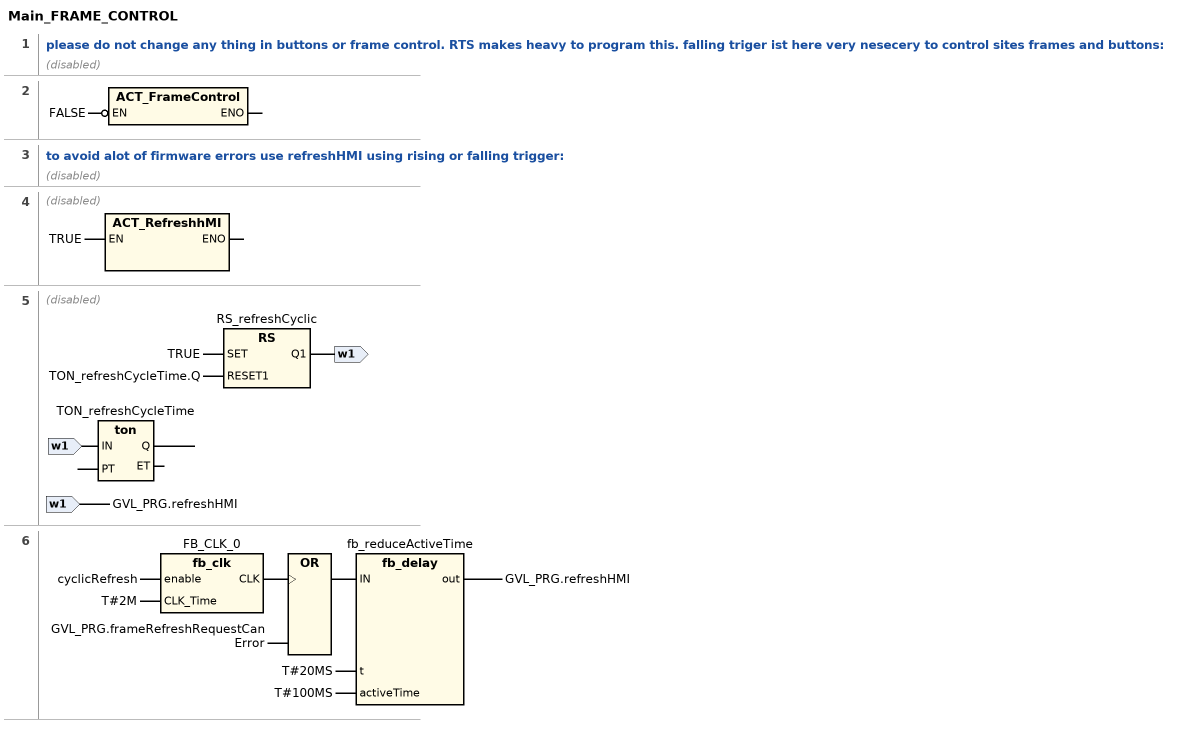
// NETWORK 1 (disabled)
// label: please do not change any thing in buttons or frame control. RTS makes heavy to program this. falling triger ist here very nesecery to control sites frames and buttons

// NETWORK 2
IF NOT FALSE THEN ACT_FrameControl(); END_IF

// NETWORK 3 (disabled)
// label: to avoid alot of firmware errors use refreshHMI using rising or falling trigger

// NETWORK 4 (disabled)
// ACT_RefreshhMI();

// NETWORK 5 (disabled)
// RS_refreshCyclic(SET := TRUE, RESET1 := TON_refreshCycleTime.Q); // RS
// TON_refreshCycleTime(IN := RS_refreshCyclic.Q1); // ton
// GVL_PRG.refreshHMI := RS_refreshCyclic.Q1;

// NETWORK 6
FB_CLK_0(enable := cyclicRefresh, CLK_Time := T#2M); // fb_clk
_rt1(CLK := FB_CLK_0.CLK);
fb_reduceActiveTime(IN := _rt1.Q OR GVL_PRG.frameRefreshRequestCanError, t := T#20MS, activeTime := T#100MS); // fb_delay
GVL_PRG.refreshHMI := fb_reduceActiveTime.out;

ACTION ACT_FrameControl:
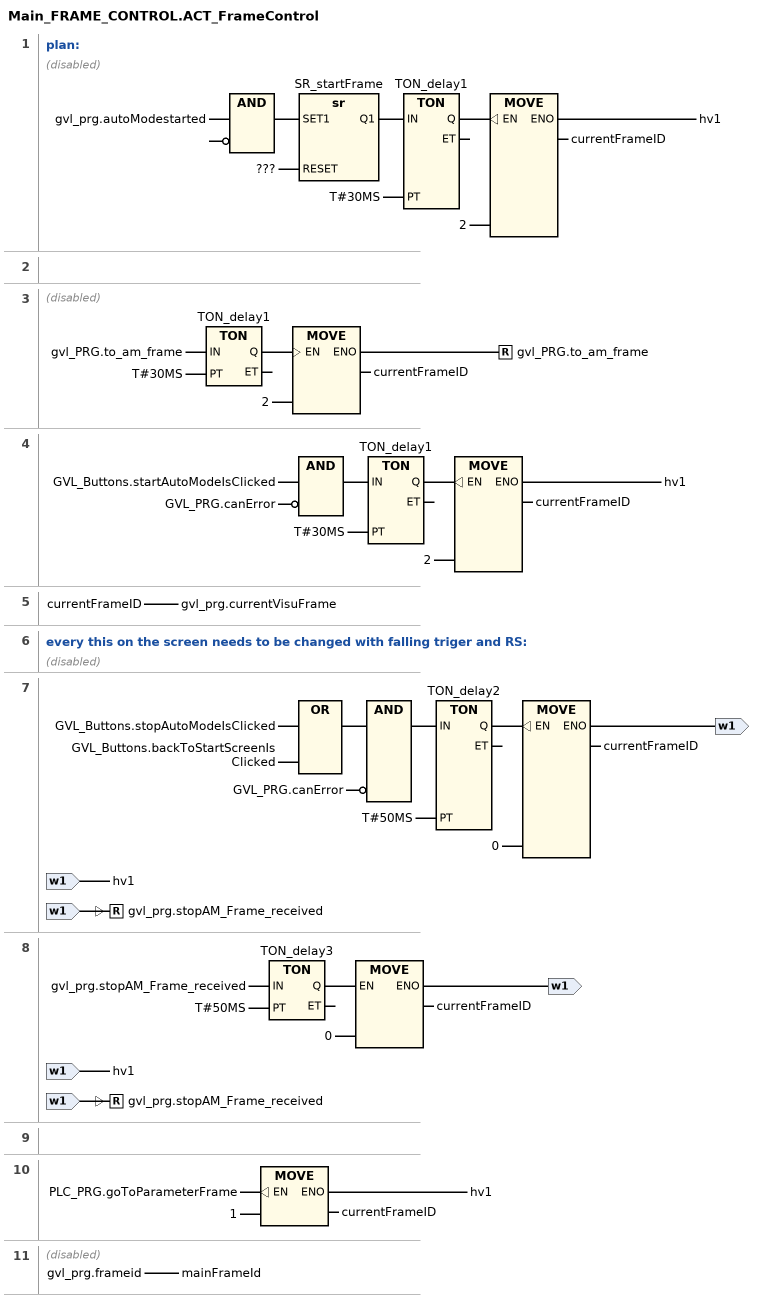
// NETWORK 1 (disabled)
// label: plan
// SR_startFrame(SET1 := gvl_prg.autoModestarted AND ???); // sr
// TON_delay1(IN := SR_startFrame.Q1, PT := T#30MS); // TON
// _ft1(CLK := TON_delay1.Q);
// _w1 := _ft1.Q;
// IF _w1 THEN currentFrameID := 2; END_IF
// hv1 := _w1;

// NETWORK 2

// NETWORK 3 (disabled)
// TON_delay1(IN := gvl_PRG.to_am_frame, PT := T#30MS); // TON
// _rt2(CLK := TON_delay1.Q);
// _w2 := _rt2.Q;
// IF _w2 THEN currentFrameID := 2; END_IF
// gvl_PRG.to_am_frame R= _w2;

// NETWORK 4
TON_delay1(IN := GVL_Buttons.startAutoModeIsClicked AND NOT GVL_PRG.canError, PT := T#30MS); // TON
_ft2(CLK := TON_delay1.Q);
_w3 := _ft2.Q;
IF _w3 THEN currentFrameID := 2; END_IF
hv1 := _w3;

// NETWORK 5
gvl_prg.currentVisuFrame := currentFrameID;

// NETWORK 6 (disabled)
// label: every this on the screen needs to be changed with falling triger and RS

// NETWORK 7
TON_delay2(IN := (GVL_Buttons.stopAutoModeIsClicked OR GVL_Buttons.backToStartScreenIsClicked) AND NOT GVL_PRG.canError, PT := T#50MS); // TON
_ft3(CLK := TON_delay2.Q);
_w4 := _ft3.Q;
IF _w4 THEN currentFrameID := 0; END_IF
hv1 := _w4;
_rt3(CLK := _w4);
gvl_prg.stopAM_Frame_received R= _rt3.Q;

// NETWORK 8
TON_delay3(IN := gvl_prg.stopAM_Frame_received, PT := T#50MS); // TON
_w5 := TON_delay3.Q;
IF _w5 THEN currentFrameID := 0; END_IF
hv1 := _w5;
_rt4(CLK := _w5);
gvl_prg.stopAM_Frame_received R= _rt4.Q;

// NETWORK 9

// NETWORK 10
_ft4(CLK := PLC_PRG.goToParameterFrame);
_w6 := _ft4.Q;
IF _w6 THEN currentFrameID := 1; END_IF
hv1 := _w6;

// NETWORK 11 (disabled)
// mainFrameId := gvl_prg.frameid;
END_ACTION

ACTION ACT_RefreshhMI:
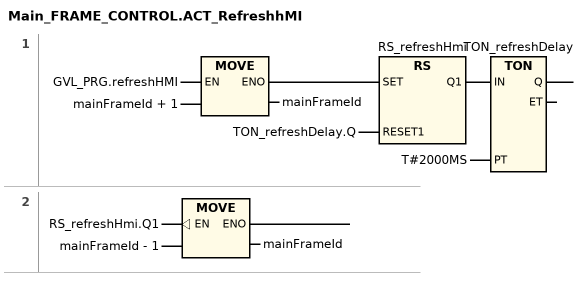
// NETWORK 1
_w7 := GVL_PRG.refreshHMI;
IF _w7 THEN mainFrameId := mainFrameId + 1; END_IF
RS_refreshHmi(SET := _w7, RESET1 := TON_refreshDelay.Q); // RS
TON_refreshDelay(IN := RS_refreshHmi.Q1, PT := T#2000MS); // TON

// NETWORK 2
_ft5(CLK := RS_refreshHmi.Q1);
IF _ft5.Q THEN mainFrameId := mainFrameId - 1; END_IF
END_ACTION

END_PROGRAM

// Device/Application/functions/fb_delay
// to delay signal and make edge signal active for a while
FUNCTION_BLOCK fb_delay 
VAR
	
	RS_1: RS;
	TON_1: TON;
	RS_2: RS;
	TON_2: TON;
END_VAR
VAR_INPUT
	IN: BOOL;
	t : TIME; 
	activeTime : TIME := T#200MS;
END_VAR

VAR_OUTPUT
	out : BOOL; // 200ms active
END_VAR

